Yaskawa INFORM job: A_ROOF_SIDE_0617_2_PAINT_20.JBI

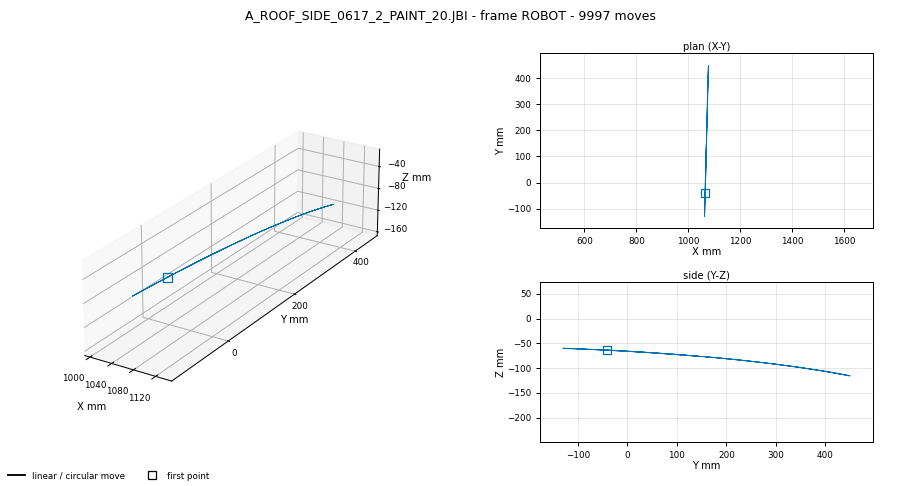
[picture p0: tool path of A_ROOF_SIDE_0617_2_PAINT_20.JBI in frame ROBOT, 9997 of 9997 moves have a stored position in this frame; points joined in program order, loops and branches not executed]
/JOB
//NAME A_ROOF_SIDE_0617_2_PAINT20
//POS
///NPOS 9997,0,0,0,0,0
///TOOL 1
///USER 0
///POSTYPE ROBOT
///RECTAN
///RCONF 1,0,0,0,0,0,0,0,0,0,0,0,0,0,0,0,0,0,0,0,0,0,0,0
C00000=1065.238,-41.066,-63.306,172.043,25.309,154.670
C00001=1065.244,-40.817,-63.319,172.044,25.312,154.670
C00002=1065.251,-40.567,-63.331,172.046,25.313,154.670
C00003=1065.257,-40.317,-63.343,172.047,25.316,154.670
C00004=1065.263,-40.068,-63.356,172.049,25.318,154.670
C00005=1065.269,-39.818,-63.369,172.050,25.320,154.671
C00006=1065.275,-39.568,-63.382,172.052,25.322,154.671
C00007=1065.281,-39.319,-63.394,172.053,25.324,154.671
C00008=1065.288,-39.070,-63.407,172.055,25.327,154.671
C00009=1065.294,-38.820,-63.420,172.056,25.328,154.671
C00010=1065.299,-38.570,-63.432,172.058,25.331,154.672
C00011=1065.305,-38.321,-63.445,172.059,25.332,154.672
C00012=1065.311,-38.071,-63.458,172.061,25.335,154.672
C00013=1065.317,-37.822,-63.471,172.063,25.337,154.672
C00014=1065.323,-37.572,-63.483,172.065,25.339,154.673
C00015=1065.329,-37.322,-63.496,172.066,25.342,154.673
C00016=1065.335,-37.073,-63.509,172.068,25.344,154.673
C00017=1065.341,-36.823,-63.522,172.069,25.346,154.673
C00018=1065.347,-36.573,-63.534,172.071,25.348,154.673
C00019=1065.353,-36.324,-63.548,172.072,25.350,154.674
C00020=1065.359,-36.074,-63.560,172.074,25.352,154.674
C00021=1065.365,-35.825,-63.573,172.075,25.355,154.674
C00022=1065.371,-35.575,-63.586,172.077,25.357,154.674
C00023=1065.378,-35.326,-63.599,172.078,25.359,154.675
C00024=1065.383,-35.076,-63.612,172.080,25.361,154.675
C00025=1065.390,-34.827,-63.625,172.081,25.363,154.675
C00026=1065.396,-34.577,-63.638,172.083,25.366,154.675
C00027=1065.402,-34.299,-63.652,172.084,25.368,154.676
C00028=1065.409,-34.021,-63.666,172.085,25.371,154.676
C00029=1065.416,-33.744,-63.680,172.088,25.373,154.676
C00030=1065.423,-33.466,-63.696,172.089,25.376,154.676
C00031=1065.429,-33.216,-63.708,172.091,25.377,154.677
C00032=1065.435,-32.967,-63.721,172.092,25.380,154.677
C00033=1065.441,-32.717,-63.734,172.094,25.382,154.677
C00034=1065.447,-32.468,-63.747,172.095,25.384,154.677
C00035=1065.453,-32.218,-63.760,172.097,25.386,154.677
C00036=1065.459,-31.969,-63.773,172.098,25.389,154.678
C00037=1065.465,-31.719,-63.786,172.100,25.391,154.678
C00038=1065.471,-31.470,-63.799,172.101,25.393,154.678
C00039=1065.477,-31.220,-63.811,172.103,25.395,154.678
C00040=1065.483,-30.970,-63.825,172.104,25.397,154.679
C00041=1065.490,-30.721,-63.838,172.106,25.400,154.679
C00042=1065.496,-30.471,-63.851,172.107,25.402,154.679
C00043=1065.502,-30.222,-63.864,172.109,25.404,154.679
C00044=1065.508,-29.971,-63.877,172.110,25.406,154.680
C00045=1065.514,-29.722,-63.890,172.112,25.409,154.680
C00046=1065.521,-29.473,-63.903,172.113,25.410,154.680
C00047=1065.526,-29.223,-63.916,172.115,25.413,154.680
C00048=1065.532,-28.973,-63.930,172.116,25.415,154.681
C00049=1065.538,-28.724,-63.943,172.117,25.417,154.681
C00050=1065.544,-28.474,-63.956,172.119,25.419,154.681
C00051=1065.550,-28.225,-63.969,172.121,25.422,154.681
C00052=1065.557,-27.976,-63.982,172.122,25.424,154.682
C00053=1065.563,-27.725,-63.995,172.123,25.426,154.682
C00054=1065.569,-27.476,-64.008,172.125,25.428,154.682
C00055=1065.576,-27.227,-64.022,172.126,25.430,154.682
C00056=1065.581,-26.977,-64.034,172.129,25.433,154.682
C00057=1065.588,-26.727,-64.047,172.130,25.435,154.683
C00058=1065.593,-26.478,-64.061,172.132,25.438,154.683
C00059=1065.599,-26.229,-64.074,172.133,25.440,154.683
C00060=1065.605,-25.979,-64.087,172.135,25.442,154.684
C00061=1065.611,-25.729,-64.101,172.136,25.444,154.684
C00062=1065.618,-25.479,-64.115,172.138,25.447,154.684
C00063=1065.624,-25.230,-64.128,172.139,25.449,154.684
C00064=1065.630,-24.980,-64.140,172.141,25.451,154.684
C00065=1065.635,-24.731,-64.154,172.142,25.454,154.685
C00066=1065.641,-24.481,-64.167,172.143,25.456,154.685
C00067=1065.648,-24.232,-64.181,172.145,25.458,154.685
C00068=1065.653,-23.982,-64.194,172.146,25.461,154.686
C00069=1065.659,-23.733,-64.207,172.148,25.463,154.686
C00070=1065.666,-23.483,-64.221,172.149,25.465,154.686
C00071=1065.671,-23.233,-64.235,172.151,25.468,154.686
C00072=1065.677,-22.984,-64.248,172.152,25.470,154.687
C00073=1065.684,-22.734,-64.261,172.154,25.472,154.687
C00074=1065.689,-22.484,-64.274,172.155,25.474,154.687
C00075=1065.695,-22.235,-64.288,172.157,25.477,154.687
C00076=1065.702,-21.985,-64.301,172.158,25.479,154.688
C00077=1065.707,-21.735,-64.315,172.160,25.481,154.688
C00078=1065.714,-21.486,-64.328,172.161,25.484,154.688
C00079=1065.720,-21.237,-64.342,172.163,25.486,154.688
C00080=1065.725,-20.987,-64.356,172.164,25.488,154.689
C00081=1065.731,-20.738,-64.369,172.165,25.491,154.689
C00082=1065.738,-20.488,-64.382,172.167,25.493,154.689
C00083=1065.743,-20.238,-64.396,172.168,25.495,154.689
C00084=1065.750,-19.989,-64.409,172.170,25.498,154.690
C00085=1065.756,-19.739,-64.422,172.171,25.500,154.690
C00086=1065.761,-19.490,-64.436,172.173,25.502,154.690
C00087=1065.768,-19.240,-64.450,172.174,25.505,154.691
C00088=1065.774,-18.991,-64.463,172.176,25.507,154.691
C00089=1065.780,-18.741,-64.477,172.177,25.509,154.691
C00090=1065.786,-18.492,-64.490,172.179,25.512,154.691
C00091=1065.793,-18.213,-64.505,172.180,25.514,154.692
C00092=1065.800,-17.934,-64.520,172.181,25.516,154.692
C00093=1065.807,-17.656,-64.536,172.184,25.520,154.692
C00094=1065.813,-17.377,-64.551,172.185,25.522,154.692
C00095=1065.820,-17.128,-64.565,172.187,25.524,154.693
C00096=1065.826,-16.879,-64.578,172.188,25.527,154.693
C00097=1065.832,-16.629,-64.592,172.190,25.529,154.693
C00098=1065.838,-16.379,-64.605,172.191,25.531,154.694
C00099=1065.844,-16.130,-64.619,172.192,25.534,154.694
C00100=1065.850,-15.881,-64.632,172.194,25.536,154.694
C00101=1065.857,-15.631,-64.646,172.195,25.538,154.694
C00102=1065.862,-15.381,-64.660,172.197,25.541,154.695
C00103=1065.868,-15.132,-64.673,172.198,25.543,154.695
C00104=1065.874,-14.881,-64.687,172.200,25.545,154.695
C00105=1065.881,-14.632,-64.701,172.201,25.548,154.695
C00106=1065.886,-14.383,-64.715,172.203,25.550,154.696
C00107=1065.893,-14.134,-64.729,172.204,25.552,154.696
C00108=1065.899,-13.884,-64.743,172.206,25.555,154.696
C00109=1065.904,-13.634,-64.757,172.207,25.557,154.697
C00110=1065.910,-13.385,-64.770,172.209,25.560,154.697
C00111=1065.916,-13.135,-64.784,172.210,25.562,154.697
C00112=1065.923,-12.885,-64.797,172.211,25.565,154.697
C00113=1065.928,-12.636,-64.811,172.213,25.567,154.698
C00114=1065.934,-12.387,-64.826,172.214,25.569,154.698
C00115=1065.940,-12.138,-64.839,172.216,25.572,154.698
C00116=1065.946,-11.887,-64.853,172.217,25.574,154.699
C00117=1065.953,-11.638,-64.867,172.219,25.576,154.699
C00118=1065.958,-11.388,-64.880,172.220,25.579,154.699
C00119=1065.964,-11.139,-64.895,172.221,25.582,154.699
C00120=1065.971,-10.889,-64.909,172.223,25.584,154.700
C00121=1065.976,-10.640,-64.923,172.224,25.586,154.700
C00122=1065.983,-10.390,-64.936,172.226,25.589,154.700
C00123=1065.988,-10.140,-64.950,172.227,25.591,154.701
C00124=1065.994,-9.891,-64.965,172.229,25.593,154.701
C00125=1066.001,-9.641,-64.978,172.230,25.596,154.701
C00126=1066.006,-9.392,-64.992,172.232,25.599,154.701
C00127=1066.012,-9.142,-65.006,172.233,25.601,154.702
C00128=1066.019,-8.893,-65.020,172.234,25.603,154.702
C00129=1066.025,-8.643,-65.034,172.236,25.606,154.702
C00130=1066.031,-8.394,-65.047,172.237,25.608,154.703
C00131=1066.037,-8.144,-65.062,172.239,25.610,154.703
C00132=1066.043,-7.895,-65.076,172.240,25.613,154.703
C00133=1066.049,-7.646,-65.090,172.242,25.616,154.703
C00134=1066.055,-7.396,-65.105,172.243,25.618,154.704
C00135=1066.061,-7.146,-65.118,172.245,25.620,154.704
C00136=1066.067,-6.896,-65.132,172.246,25.623,154.704
C00137=1066.073,-6.647,-65.147,172.247,25.625,154.705
C00138=1066.079,-6.398,-65.160,172.249,25.627,154.705
C00139=1066.086,-6.148,-65.174,172.250,25.630,154.705
C00140=1066.091,-5.899,-65.189,172.252,25.633,154.706
C00141=1066.097,-5.649,-65.203,172.253,25.635,154.706
C00142=1066.104,-5.399,-65.216,172.255,25.637,154.706
C00143=1066.110,-5.150,-65.231,172.256,25.640,154.706
C00144=1066.115,-4.900,-65.245,172.258,25.642,154.707
C00145=1066.122,-4.652,-65.259,172.259,25.644,154.707
C00146=1066.128,-4.401,-65.273,172.260,25.647,154.707
C00147=1066.134,-4.152,-65.287,172.262,25.649,154.708
C00148=1066.141,-3.902,-65.301,172.263,25.652,154.708
C00149=1066.146,-3.653,-65.315,172.265,25.654,154.708
C00150=1066.153,-3.403,-65.330,172.266,25.656,154.708
C00151=1066.158,-3.154,-65.344,172.268,25.659,154.709
C00152=1066.164,-2.905,-65.359,172.269,25.662,154.709
C00153=1066.171,-2.655,-65.372,172.271,25.664,154.709
C00154=1066.176,-2.405,-65.386,172.272,25.666,154.710
C00155=1066.182,-2.125,-65.403,172.273,25.669,154.710
C00156=1066.189,-1.844,-65.419,172.275,25.672,154.710
C00157=1066.196,-1.565,-65.435,172.277,25.675,154.711
C00158=1066.202,-1.285,-65.451,172.278,25.678,154.711
C00159=1066.208,-1.035,-65.465,172.280,25.681,154.711
C00160=1066.214,-0.786,-65.480,172.281,25.683,154.712
C00161=1066.220,-0.536,-65.494,172.283,25.685,154.712
C00162=1066.226,-0.286,-65.509,172.284,25.688,154.712
C00163=1066.232,-0.037,-65.523,172.286,25.691,154.713
C00164=1066.238,0.213,-65.538,172.287,25.693,154.713
C00165=1066.245,0.461,-65.552,172.288,25.696,154.713
C00166=1066.250,0.711,-65.566,172.290,25.698,154.713
C00167=1066.256,0.961,-65.581,172.291,25.700,154.714
C00168=1066.262,1.210,-65.595,172.293,25.703,154.714
C00169=1066.268,1.460,-65.610,172.294,25.706,154.714
C00170=1066.274,1.709,-65.624,172.296,25.708,154.715
C00171=1066.280,1.959,-65.638,172.297,25.711,154.715
C00172=1066.286,2.208,-65.653,172.298,25.713,154.715
C00173=1066.292,2.458,-65.667,172.300,25.716,154.716
C00174=1066.298,2.707,-65.682,172.301,25.719,154.716
C00175=1066.304,2.957,-65.697,172.303,25.721,154.716
C00176=1066.310,3.207,-65.711,172.304,25.723,154.717
C00177=1066.316,3.456,-65.725,172.305,25.726,154.717
C00178=1066.322,3.705,-65.740,172.307,25.728,154.717
C00179=1066.328,3.955,-65.754,172.308,25.731,154.717
C00180=1066.334,4.204,-65.769,172.310,25.734,154.718
C00181=1066.340,4.454,-65.784,172.311,25.736,154.718
C00182=1066.346,4.704,-65.798,172.313,25.738,154.718
C00183=1066.352,4.953,-65.813,172.314,25.741,154.719
C00184=1066.358,5.202,-65.827,172.316,25.744,154.719
C00185=1066.364,5.452,-65.842,172.317,25.746,154.719
C00186=1066.370,5.701,-65.856,172.318,25.749,154.720
C00187=1066.376,5.951,-65.871,172.320,25.751,154.720
C00188=1066.382,6.200,-65.886,172.320,25.754,154.720
C00189=1066.388,6.450,-65.900,172.322,25.756,154.721
C00190=1066.394,6.699,-65.914,172.323,25.758,154.721
C00191=1066.400,6.949,-65.929,172.325,25.761,154.721
C00192=1066.406,7.199,-65.944,172.326,25.764,154.722
C00193=1066.412,7.448,-65.959,172.328,25.766,154.722
C00194=1066.417,7.698,-65.974,172.329,25.769,154.722
C00195=1066.423,7.947,-65.988,172.330,25.771,154.723
C00196=1066.430,8.197,-66.003,172.332,25.773,154.723
C00197=1066.435,8.446,-66.018,172.333,25.776,154.723
C00198=1066.442,8.695,-66.033,172.335,25.779,154.724
C00199=1066.448,8.946,-66.047,172.336,25.781,154.724
C00200=1066.454,9.195,-66.062,172.337,25.784,154.724
C00201=1066.460,9.444,-66.076,172.339,25.786,154.725
C00202=1066.466,9.694,-66.091,172.340,25.789,154.725
C00203=1066.472,9.943,-66.106,172.342,25.791,154.725
C00204=1066.479,10.193,-66.121,172.343,25.794,154.725
C00205=1066.484,10.441,-66.136,172.345,25.797,154.726
C00206=1066.490,10.692,-66.150,172.346,25.799,154.726
C00207=1066.497,10.941,-66.165,172.348,25.801,154.726
C00208=1066.503,11.190,-66.179,172.349,25.804,154.727
C00209=1066.509,11.440,-66.194,172.350,25.807,154.727
C00210=1066.515,11.690,-66.209,172.352,25.809,154.727
C00211=1066.520,11.939,-66.224,172.353,25.812,154.728
C00212=1066.527,12.189,-66.239,172.355,25.814,154.728
C00213=1066.533,12.438,-66.254,172.356,25.816,154.728
C00214=1066.539,12.687,-66.269,172.358,25.819,154.729
C00215=1066.545,12.937,-66.284,172.359,25.822,154.729
C00216=1066.552,13.187,-66.299,172.360,25.824,154.729
C00217=1066.558,13.435,-66.313,172.362,25.827,154.730
C00218=1066.564,13.685,-66.328,172.363,25.829,154.730
C00219=1066.571,13.967,-66.345,172.365,25.832,154.730
C00220=1066.577,14.249,-66.362,172.366,25.835,154.731
C00221=1066.584,14.532,-66.378,172.368,25.838,154.731
C00222=1066.591,14.813,-66.396,172.370,25.841,154.731
C00223=1066.597,15.063,-66.411,172.371,25.843,154.732
C00224=1066.603,15.312,-66.426,172.373,25.846,154.732
C00225=1066.609,15.562,-66.441,172.374,25.849,154.732
C00226=1066.615,15.812,-66.456,172.375,25.851,154.733
C00227=1066.621,16.061,-66.471,172.377,25.854,154.733
C00228=1066.627,16.310,-66.486,172.378,25.856,154.733
C00229=1066.633,16.560,-66.501,172.380,25.859,154.734
C00230=1066.638,16.809,-66.516,172.381,25.861,154.734
C00231=1066.645,17.059,-66.531,172.382,25.864,154.734
C00232=1066.651,17.308,-66.546,172.384,25.867,154.735
C00233=1066.656,17.558,-66.561,172.385,25.869,154.735
C00234=1066.663,17.807,-66.576,172.387,25.872,154.735
C00235=1066.669,18.057,-66.591,172.388,25.875,154.736
C00236=1066.674,18.306,-66.607,172.390,25.877,154.736
C00237=1066.681,18.555,-66.622,172.391,25.880,154.736
C00238=1066.687,18.805,-66.637,172.392,25.882,154.737
C00239=1066.693,19.055,-66.652,172.393,25.885,154.737
C00240=1066.699,19.304,-66.667,172.394,25.887,154.737
C00241=1066.705,19.554,-66.682,172.396,25.890,154.738
C00242=1066.711,19.803,-66.698,172.397,25.892,154.738
C00243=1066.717,20.053,-66.713,172.399,25.895,154.738
C00244=1066.723,20.302,-66.728,172.400,25.897,154.739
C00245=1066.729,20.552,-66.743,172.401,25.900,154.739
C00246=1066.735,20.801,-66.758,172.403,25.903,154.739
C00247=1066.740,21.050,-66.774,172.404,25.906,154.740
C00248=1066.747,21.299,-66.789,172.406,25.908,154.740
C00249=1066.752,21.549,-66.804,172.407,25.911,154.740
C00250=1066.759,21.799,-66.819,172.409,25.913,154.741
C00251=1066.764,22.048,-66.835,172.410,25.916,154.741
C00252=1066.771,22.297,-66.850,172.411,25.918,154.741
C00253=1066.776,22.547,-66.866,172.413,25.921,154.742
C00254=1066.783,22.797,-66.881,172.414,25.923,154.742
C00255=1066.789,23.045,-66.896,172.416,25.926,154.742
C00256=1066.794,23.295,-66.912,172.417,25.929,154.743
C00257=1066.801,23.545,-66.927,172.419,25.932,154.743
C00258=1066.806,23.795,-66.942,172.420,25.934,154.743
C00259=1066.812,24.043,-66.957,172.421,25.937,154.744
C00260=1066.818,24.293,-66.973,172.423,25.940,154.744
C00261=1066.824,24.543,-66.988,172.424,25.942,154.744
C00262=1066.830,24.792,-67.004,172.426,25.945,154.745
C00263=1066.837,25.042,-67.019,172.427,25.947,154.745
C00264=1066.842,25.291,-67.034,172.428,25.950,154.745
C00265=1066.849,25.540,-67.050,172.430,25.952,154.746
C00266=1066.854,25.790,-67.065,172.431,25.955,154.746
C00267=1066.861,26.040,-67.080,172.433,25.958,154.746
C00268=1066.866,26.289,-67.097,172.434,25.960,154.747
C00269=1066.872,26.538,-67.111,172.436,25.963,154.747
C00270=1066.878,26.788,-67.127,172.437,25.966,154.747
C00271=1066.885,27.037,-67.142,172.438,25.968,154.748
C00272=1066.890,27.287,-67.158,172.440,25.971,154.748
C00273=1066.897,27.536,-67.174,172.441,25.974,154.749
C00274=1066.902,27.785,-67.189,172.443,25.976,154.749
C00275=1066.908,28.035,-67.205,172.444,25.979,154.749
C00276=1066.914,28.284,-67.220,172.446,25.981,154.749
C00277=1066.920,28.534,-67.236,172.446,25.984,154.750
C00278=1066.927,28.783,-67.251,172.447,25.986,154.750
C00279=1066.933,29.033,-67.267,172.449,25.989,154.751
C00280=1066.938,29.282,-67.283,172.450,25.992,154.751
C00281=1066.944,29.531,-67.298,172.452,25.994,154.751
C00282=1066.950,29.781,-67.314,172.453,25.997,154.752
C00283=1066.957,30.064,-67.331,172.455,26.000,154.752
C00284=1066.964,30.348,-67.350,172.457,26.003,154.752
C00285=1066.971,30.631,-67.367,172.458,26.006,154.753
C00286=1066.977,30.914,-67.385,172.459,26.009,154.753
C00287=1066.983,31.164,-67.400,172.461,26.012,154.754
C00288=1066.989,31.414,-67.417,172.462,26.014,154.754
C00289=1066.995,31.663,-67.433,172.464,26.017,154.754
C00290=1067.001,31.913,-67.448,172.465,26.020,154.755
C00291=1067.006,32.161,-67.464,172.467,26.022,154.755
C00292=1067.012,32.411,-67.479,172.468,26.025,154.755
C00293=1067.019,32.660,-67.495,172.469,26.028,154.756
C00294=1067.024,32.910,-67.510,172.471,26.030,154.756
C00295=1067.030,33.160,-67.527,172.472,26.033,154.756
C00296=1067.036,33.409,-67.543,172.474,26.035,154.757
C00297=1067.043,33.659,-67.558,172.475,26.038,154.757
C00298=1067.049,33.908,-67.574,172.476,26.041,154.757
C00299=1067.055,34.157,-67.590,172.478,26.043,154.758
C00300=1067.060,34.407,-67.606,172.479,26.046,154.758
C00301=1067.066,34.656,-67.621,172.481,26.049,154.758
C00302=1067.072,34.906,-67.637,172.482,26.052,154.759
C00303=1067.078,35.155,-67.653,172.484,26.054,154.759
C00304=1067.085,35.404,-67.669,172.485,26.057,154.759
C00305=1067.091,35.653,-67.685,172.486,26.060,154.760
C00306=1067.096,35.903,-67.701,172.488,26.062,154.760
C00307=1067.102,36.153,-67.717,172.489,26.065,154.761
C00308=1067.108,36.402,-67.733,172.491,26.068,154.761
C00309=1067.115,36.652,-67.748,172.492,26.070,154.761
C00310=1067.120,36.901,-67.764,172.494,26.073,154.762
C00311=1067.126,37.150,-67.780,172.495,26.075,154.762
C00312=1067.132,37.400,-67.796,172.496,26.078,154.762
C00313=1067.139,37.649,-67.812,172.498,26.081,154.763
C00314=1067.145,37.899,-67.828,172.499,26.083,154.763
C00315=1067.151,38.148,-67.844,172.501,26.086,154.763
C00316=1067.156,38.398,-67.860,172.502,26.089,154.764
C00317=1067.162,38.647,-67.876,172.503,26.091,154.764
C00318=1067.168,38.896,-67.892,172.504,26.094,154.764
C00319=1067.174,39.145,-67.908,172.505,26.097,154.765
C00320=1067.179,39.395,-67.924,172.507,26.099,154.765
C00321=1067.185,39.645,-67.940,172.508,26.102,154.766
C00322=1067.191,39.894,-67.956,172.510,26.105,154.766
C00323=1067.197,40.143,-67.972,172.511,26.107,154.766
C00324=1067.203,40.393,-67.989,172.512,26.110,154.767
C00325=1067.209,40.642,-68.005,172.514,26.113,154.767
C00326=1067.216,40.891,-68.021,172.515,26.115,154.767
C00327=1067.221,41.141,-68.036,172.517,26.118,154.768
C00328=1067.227,41.391,-68.052,172.518,26.121,154.768
C00329=1067.233,41.640,-68.069,172.520,26.123,154.768
C00330=1067.239,41.889,-68.085,172.521,26.126,154.769
C00331=1067.245,42.139,-68.101,172.522,26.129,154.769
C00332=1067.251,42.388,-68.117,172.524,26.131,154.769
C00333=1067.257,42.637,-68.134,172.525,26.134,154.770
C00334=1067.263,42.887,-68.150,172.527,26.137,154.770
C00335=1067.269,43.136,-68.166,172.528,26.139,154.771
C00336=1067.275,43.385,-68.182,172.530,26.142,154.771
C00337=1067.280,43.635,-68.198,172.531,26.145,154.771
C00338=1067.286,43.885,-68.214,172.532,26.148,154.772
C00339=1067.292,44.134,-68.231,172.534,26.150,154.772
C00340=1067.298,44.384,-68.247,172.535,26.153,154.772
C00341=1067.304,44.633,-68.264,172.537,26.156,154.773
C00342=1067.310,44.882,-68.280,172.538,26.159,154.773
C00343=1067.315,45.132,-68.296,172.539,26.161,154.773
C00344=1067.321,45.381,-68.312,172.541,26.164,154.774
C00345=1067.327,45.631,-68.329,172.542,26.167,154.774
C00346=1067.333,45.880,-68.346,172.544,26.170,154.775
C00347=1067.340,46.163,-68.364,172.545,26.173,154.775
C00348=1067.346,46.447,-68.383,172.546,26.175,154.775
C00349=1067.352,46.730,-68.402,172.548,26.179,154.776
C00350=1067.360,47.013,-68.420,172.550,26.182,154.776
C00351=1067.365,47.263,-68.437,172.551,26.185,154.777
C00352=1067.371,47.512,-68.453,172.553,26.187,154.777
C00353=1067.377,47.761,-68.470,172.554,26.190,154.777
C00354=1067.383,48.011,-68.486,172.556,26.193,154.778
C00355=1067.389,48.260,-68.502,172.557,26.196,154.778
C00356=1067.394,48.510,-68.519,172.559,26.198,154.778
C00357=1067.400,48.759,-68.535,172.560,26.201,154.779
C00358=1067.406,49.008,-68.551,172.561,26.204,154.779
C00359=1067.412,49.258,-68.568,172.563,26.207,154.780
C00360=1067.417,49.507,-68.585,172.563,26.209,154.780
C00361=1067.423,49.756,-68.602,172.565,26.211,154.780
C00362=1067.429,50.005,-68.618,172.566,26.214,154.781
C00363=1067.436,50.255,-68.634,172.567,26.217,154.781
C00364=1067.441,50.505,-68.651,172.569,26.220,154.781
C00365=1067.447,50.754,-68.668,172.570,26.222,154.782
C00366=1067.453,51.004,-68.684,172.572,26.225,154.782
C00367=1067.459,51.253,-68.701,172.573,26.228,154.783
C00368=1067.464,51.502,-68.718,172.575,26.230,154.783
C00369=1067.470,51.752,-68.734,172.576,26.233,154.783
C00370=1067.476,52.001,-68.750,172.577,26.236,154.784
C00371=1067.482,52.250,-68.766,172.579,26.239,154.784
C00372=1067.488,52.499,-68.784,172.580,26.241,154.784
C00373=1067.494,52.749,-68.801,172.582,26.244,154.785
C00374=1067.500,52.999,-68.817,172.583,26.247,154.785
C00375=1067.506,53.248,-68.833,172.584,26.250,154.786
C00376=1067.512,53.497,-68.851,172.586,26.252,154.786
C00377=1067.518,53.746,-68.867,172.587,26.255,154.786
C00378=1067.524,53.996,-68.883,172.589,26.258,154.787
C00379=1067.530,54.245,-68.899,172.590,26.260,154.787
C00380=1067.536,54.495,-68.917,172.592,26.263,154.787
C00381=1067.542,54.744,-68.934,172.593,26.266,154.788
C00382=1067.548,54.994,-68.950,172.594,26.269,154.788
C00383=1067.553,55.243,-68.967,172.596,26.271,154.788
C00384=1067.559,55.492,-68.984,172.597,26.274,154.789
C00385=1067.565,55.741,-69.000,172.599,26.277,154.789
C00386=1067.572,55.991,-69.017,172.600,26.279,154.789
C00387=1067.577,56.240,-69.034,172.602,26.282,154.790
C00388=1067.583,56.490,-69.050,172.603,26.285,154.790
C00389=1067.589,56.738,-69.067,172.604,26.288,154.791
C00390=1067.595,56.988,-69.084,172.606,26.290,154.791
C00391=1067.601,57.238,-69.101,172.607,26.293,154.791
C00392=1067.607,57.487,-69.118,172.609,26.296,154.792
C00393=1067.613,57.737,-69.135,172.610,26.298,154.792
C00394=1067.619,57.986,-69.151,172.612,26.301,154.792
C00395=1067.625,58.235,-69.168,172.613,26.304,154.793
C00396=1067.631,58.485,-69.185,172.615,26.306,154.793
C00397=1067.637,58.734,-69.202,172.616,26.309,154.793
C00398=1067.643,58.983,-69.218,172.617,26.312,154.794
C00399=1067.649,59.233,-69.236,172.619,26.314,154.794
C00400=1067.655,59.482,-69.253,172.620,26.317,154.795
C00401=1067.661,59.732,-69.269,172.622,26.320,154.795
C00402=1067.666,59.981,-69.286,172.623,26.322,154.795
C00403=1067.673,60.231,-69.303,172.625,26.325,154.796
C00404=1067.679,60.479,-69.320,172.626,26.328,154.796
C00405=1067.684,60.729,-69.337,172.627,26.330,154.796
C00406=1067.691,60.978,-69.354,172.629,26.333,154.797
C00407=1067.697,61.228,-69.370,172.630,26.336,154.797
C00408=1067.703,61.477,-69.388,172.632,26.338,154.797
C00409=1067.709,61.726,-69.404,172.633,26.341,154.798
C00410=1067.716,61.976,-69.422,172.635,26.344,154.798
C00411=1067.722,62.258,-69.441,172.636,26.347,154.799
C00412=1067.729,62.542,-69.460,172.637,26.349,154.799
C00413=1067.736,62.825,-69.480,172.640,26.353,154.799
C00414=1067.742,63.108,-69.499,172.641,26.355,154.800
C00415=1067.748,63.358,-69.516,172.643,26.358,154.800
C00416=1067.755,63.607,-69.533,172.644,26.361,154.801
C00417=1067.760,63.856,-69.550,172.645,26.363,154.801
C00418=1067.767,64.106,-69.567,172.647,26.366,154.801
C00419=1067.773,64.354,-69.584,172.648,26.369,154.802
C00420=1067.778,64.604,-69.601,172.650,26.371,154.802
C00421=1067.784,64.854,-69.618,172.651,26.374,154.802
C00422=1067.791,65.103,-69.635,172.653,26.377,154.803
C00423=1067.796,65.352,-69.652,172.654,26.380,154.803
C00424=1067.803,65.602,-69.670,172.655,26.382,154.803
C00425=1067.808,65.851,-69.687,172.657,26.385,154.804
C00426=1067.813,66.100,-69.704,172.658,26.388,154.804
C00427=1067.820,66.349,-69.721,172.660,26.391,154.805
C00428=1067.826,66.599,-69.739,172.661,26.393,154.805
C00429=1067.832,66.848,-69.755,172.663,26.396,154.805
C00430=1067.837,67.097,-69.773,172.664,26.399,154.806
C00431=1067.843,67.347,-69.791,172.665,26.402,154.806
C00432=1067.849,67.596,-69.807,172.667,26.404,154.806
C00433=1067.855,67.845,-69.825,172.668,26.407,154.807
C00434=1067.861,68.095,-69.842,172.670,26.410,154.807
C00435=1067.867,68.344,-69.859,172.671,26.412,154.808
C00436=1067.872,68.593,-69.876,172.673,26.415,154.808
C00437=1067.879,68.843,-69.894,172.674,26.418,154.808
C00438=1067.885,69.092,-69.911,172.675,26.420,154.809
C00439=1067.890,69.319,-69.927,172.677,26.423,154.809
C00440=1067.896,69.546,-69.943,172.677,26.425,154.809
C00441=1067.900,69.774,-69.959,172.679,26.428,154.810
C00442=1067.906,70.001,-69.974,172.680,26.430,154.810
C00443=1067.912,70.228,-69.990,172.682,26.433,154.810
C00444=1067.917,70.455,-70.006,172.683,26.435,154.811
C00445=1067.923,70.682,-70.022,172.685,26.438,154.811
C00446=1067.927,70.910,-70.038,172.685,26.440,154.811
C00447=1067.934,71.159,-70.055,172.687,26.443,154.812
C00448=1067.940,71.408,-70.073,172.688,26.445,154.812
C00449=1067.945,71.657,-70.090,172.690,26.448,154.813
C00450=1067.951,71.906,-70.108,172.691,26.451,154.813
C00451=1067.957,72.157,-70.125,172.693,26.453,154.813
C00452=1067.963,72.406,-70.142,172.694,26.456,154.814
C00453=1067.969,72.655,-70.160,172.695,26.459,154.814
C00454=1067.974,72.904,-70.178,172.697,26.462,154.814
C00455=1067.980,73.153,-70.195,172.698,26.464,154.815
C00456=1067.986,73.403,-70.213,172.700,26.467,154.815
C00457=1067.992,73.652,-70.230,172.702,26.470,154.815
C00458=1067.998,73.901,-70.248,172.704,26.473,154.816
C00459=1068.004,74.151,-70.266,172.705,26.476,154.816
C00460=1068.010,74.400,-70.283,172.706,26.478,154.817
C00461=1068.015,74.650,-70.300,172.708,26.481,154.817
C00462=1068.021,74.899,-70.318,172.709,26.484,154.817
C00463=1068.028,75.149,-70.335,172.711,26.487,154.818
C00464=1068.033,75.398,-70.353,172.712,26.489,154.818
C00465=1068.039,75.647,-70.370,172.714,26.492,154.818
C00466=1068.045,75.896,-70.388,172.715,26.495,154.819
C00467=1068.050,76.145,-70.406,172.716,26.498,154.819
C00468=1068.057,76.395,-70.424,172.718,26.500,154.819
C00469=1068.063,76.644,-70.441,172.719,26.503,154.820
C00470=1068.069,76.894,-70.459,172.721,26.505,154.820
C00471=1068.074,77.143,-70.476,172.722,26.508,154.821
C00472=1068.081,77.392,-70.494,172.724,26.511,154.821
C00473=1068.086,77.641,-70.512,172.725,26.513,154.821
C00474=1068.092,77.891,-70.531,172.727,26.516,154.822
C00475=1068.100,78.218,-70.553,172.728,26.520,154.822
C00476=1068.108,78.545,-70.577,172.730,26.523,154.823
C00477=1068.116,78.872,-70.600,172.732,26.527,154.823
C00478=1068.123,79.200,-70.623,172.734,26.530,154.824
C00479=1068.128,79.449,-70.641,172.735,26.533,154.824
C00480=1068.135,79.698,-70.659,172.737,26.536,154.825
C00481=1068.140,79.947,-70.677,172.738,26.538,154.825
C00482=1068.146,80.197,-70.695,172.739,26.541,154.825
C00483=1068.152,80.446,-70.712,172.741,26.544,154.826
C00484=1068.158,80.696,-70.730,172.742,26.547,154.826
C00485=1068.164,80.945,-70.748,172.744,26.550,154.826
C00486=1068.170,81.194,-70.766,172.746,26.553,154.827
C00487=1068.176,81.443,-70.784,172.748,26.555,154.827
C00488=1068.180,81.692,-70.802,172.749,26.558,154.827
C00489=1068.186,81.942,-70.820,172.750,26.561,154.828
C00490=1068.192,82.191,-70.838,172.752,26.564,154.828
C00491=1068.198,82.441,-70.856,172.753,26.567,154.829
C00492=1068.204,82.689,-70.874,172.755,26.569,154.829
C00493=1068.210,82.939,-70.892,172.756,26.572,154.829
C00494=1068.216,83.188,-70.909,172.758,26.574,154.830
C00495=1068.222,83.438,-70.927,172.759,26.577,154.830
C00496=1068.228,83.687,-70.946,172.761,26.580,154.831
C00497=1068.234,83.936,-70.964,172.762,26.582,154.831
C00498=1068.239,84.186,-70.982,172.763,26.585,154.831
C00499=1068.245,84.435,-71.000,172.765,26.588,154.832
C00500=1068.251,84.684,-71.018,172.766,26.591,154.832
C00501=1068.256,84.933,-71.036,172.768,26.594,154.832
C00502=1068.263,85.183,-71.054,172.769,26.596,154.833
C00503=1068.268,85.431,-71.072,172.771,26.599,154.833
C00504=1068.275,85.681,-71.090,172.772,26.602,154.834
C00505=1068.280,85.930,-71.108,172.774,26.605,154.834
C00506=1068.286,86.180,-71.126,172.775,26.607,154.834
C00507=1068.292,86.429,-71.145,172.776,26.610,154.835
C00508=1068.297,86.678,-71.162,172.778,26.612,154.835
C00509=1068.304,86.927,-71.181,172.779,26.615,154.835
C00510=1068.309,87.176,-71.199,172.781,26.618,154.836
C00511=1068.315,87.426,-71.217,172.782,26.620,154.836
C00512=1068.322,87.675,-71.235,172.784,26.623,154.837
C00513=1068.327,87.924,-71.253,172.785,26.626,154.837
C00514=1068.333,88.174,-71.271,172.787,26.628,154.837
C00515=1068.339,88.423,-71.290,172.788,26.631,154.838
C00516=1068.345,88.672,-71.307,172.790,26.634,154.838
C00517=1068.351,88.922,-71.326,172.792,26.637,154.838
C00518=1068.357,89.171,-71.344,172.793,26.639,154.839
C00519=1068.363,89.420,-71.362,172.795,26.642,154.839
C00520=1068.368,89.670,-71.381,172.796,26.645,154.839
C00521=1068.374,89.919,-71.398,172.798,26.648,154.840
C00522=1068.380,90.168,-71.417,172.799,26.650,154.840
C00523=1068.386,90.417,-71.435,172.801,26.653,154.841
C00524=1068.392,90.666,-71.453,172.802,26.656,154.841
C00525=1068.398,90.916,-71.471,172.804,26.658,154.841
C00526=1068.404,91.165,-71.490,172.805,26.661,154.842
C00527=1068.410,91.414,-71.508,172.807,26.664,154.842
C00528=1068.415,91.664,-71.527,172.808,26.667,154.842
C00529=1068.421,91.913,-71.545,172.809,26.669,154.843
C00530=1068.427,92.162,-71.564,172.811,26.672,154.843
C00531=1068.432,92.411,-71.582,172.812,26.674,154.844
C00532=1068.439,92.660,-71.600,172.814,26.677,154.844
C00533=1068.444,92.910,-71.620,172.815,26.680,154.844
C00534=1068.450,93.159,-71.637,172.817,26.683,154.845
C00535=1068.456,93.408,-71.656,172.818,26.686,154.845
C00536=1068.462,93.658,-71.674,172.819,26.689,154.846
C00537=1068.467,93.906,-71.693,172.822,26.691,154.846
C00538=1068.473,94.156,-71.712,172.823,26.694,154.846
C00539=1068.480,94.439,-71.732,172.825,26.697,154.847
C00540=1068.487,94.722,-71.753,172.826,26.700,154.847
C00541=1068.493,95.005,-71.774,172.829,26.703,154.847
C00542=1068.500,95.288,-71.795,172.830,26.706,154.848
C00543=1068.505,95.537,-71.814,172.831,26.709,154.848
C00544=1068.512,95.786,-71.832,172.833,26.712,154.849
C00545=1068.516,96.036,-71.851,172.834,26.715,154.849
C00546=1068.523,96.285,-71.869,172.836,26.717,154.849
C00547=1068.529,96.534,-71.888,172.837,26.720,154.850
C00548=1068.534,96.783,-71.906,172.839,26.723,154.850
C00549=1068.541,97.033,-71.925,172.840,26.725,154.851
C00550=1068.546,97.282,-71.944,172.842,26.728,154.851
C00551=1068.553,97.531,-71.963,172.844,26.731,154.851
C00552=1068.557,97.780,-71.981,172.845,26.734,154.852
C00553=1068.564,98.030,-71.999,172.847,26.736,154.852
C00554=1068.570,98.279,-72.019,172.848,26.739,154.852
C00555=1068.576,98.528,-72.037,172.850,26.742,154.853
C00556=1068.581,98.777,-72.055,172.851,26.744,154.853
C00557=1068.587,99.027,-72.074,172.853,26.747,154.854
C00558=1068.594,99.276,-72.093,172.854,26.750,154.854
C00559=1068.599,99.525,-72.112,172.856,26.752,154.854
C00560=1068.605,99.774,-72.130,172.857,26.755,154.855
C00561=1068.611,100.024,-72.149,172.859,26.758,154.855
C00562=1068.617,100.273,-72.167,172.860,26.761,154.855
C00563=1068.623,100.522,-72.187,172.862,26.763,154.856
C00564=1068.628,100.771,-72.205,172.863,26.766,154.856
C00565=1068.634,101.021,-72.224,172.865,26.769,154.856
C00566=1068.640,101.270,-72.242,172.867,26.772,154.857
C00567=1068.646,101.519,-72.261,172.868,26.775,154.857
C00568=1068.651,101.768,-72.280,172.870,26.777,154.858
C00569=1068.657,102.017,-72.299,172.871,26.780,154.858
C00570=1068.663,102.266,-72.318,172.873,26.782,154.858
C00571=1068.669,102.516,-72.337,172.874,26.785,154.859
C00572=1068.675,102.764,-72.356,172.876,26.788,154.859
C00573=1068.680,103.014,-72.375,172.877,26.791,154.860
C00574=1068.686,103.264,-72.393,172.879,26.793,154.860
C00575=1068.692,103.513,-72.412,172.880,26.796,154.860
C00576=1068.697,103.762,-72.431,172.881,26.799,154.861
C00577=1068.703,104.011,-72.450,172.884,26.802,154.861
C00578=1068.709,104.261,-72.469,172.885,26.805,154.861
C00579=1068.715,104.510,-72.488,172.887,26.807,154.862
C00580=1068.721,104.759,-72.507,172.888,26.810,154.862
C00581=1068.726,105.008,-72.526,172.890,26.813,154.863
C00582=1068.732,105.257,-72.545,172.891,26.815,154.863
C00583=1068.738,105.506,-72.564,172.893,26.818,154.863
C00584=1068.744,105.756,-72.583,172.894,26.820,154.864
C00585=1068.750,106.005,-72.602,172.896,26.823,154.864
C00586=1068.755,106.254,-72.621,172.897,26.826,154.864
C00587=1068.761,106.503,-72.640,172.898,26.829,154.865
C00588=1068.767,106.753,-72.659,172.901,26.832,154.865
C00589=1068.773,107.002,-72.678,172.902,26.834,154.865
C00590=1068.779,107.251,-72.697,172.904,26.837,154.866
C00591=1068.784,107.501,-72.717,172.905,26.840,154.866
C00592=1068.790,107.750,-72.736,172.907,26.843,154.867
C00593=1068.796,107.998,-72.755,172.908,26.845,154.867
C00594=1068.802,108.247,-72.774,172.910,26.848,154.867
C00595=1068.808,108.497,-72.793,172.911,26.851,154.868
C00596=1068.813,108.746,-72.813,172.913,26.853,154.868
C00597=1068.820,108.995,-72.831,172.914,26.856,154.868
C00598=1068.825,109.245,-72.850,172.917,26.859,154.869
C00599=1068.831,109.494,-72.870,172.918,26.862,154.869
C00600=1068.837,109.743,-72.889,172.919,26.864,154.870
C00601=1068.843,109.991,-72.908,172.921,26.867,154.870
C00602=1068.849,110.241,-72.927,172.922,26.869,154.870
C00603=1068.856,110.524,-72.949,172.924,26.872,154.871
C00604=1068.862,110.807,-72.971,172.926,26.876,154.871
C00605=1068.869,111.090,-72.993,172.928,26.879,154.872
C00606=1068.875,111.373,-73.015,172.930,26.882,154.872
C00607=1068.881,111.623,-73.034,172.931,26.885,154.872
C00608=1068.886,111.872,-73.053,172.933,26.887,154.873
C00609=1068.893,112.121,-73.072,172.934,26.890,154.873
C00610=1068.899,112.370,-73.092,172.936,26.893,154.874
C00611=1068.904,112.620,-73.111,172.937,26.895,154.874
C00612=1068.910,112.869,-73.130,172.939,26.898,154.874
C00613=1068.916,113.118,-73.149,172.940,26.901,154.875
C00614=1068.921,113.366,-73.169,172.943,26.903,154.875
C00615=1068.927,113.616,-73.188,172.944,26.906,154.875
C00616=1068.933,113.865,-73.207,172.946,26.909,154.876
C00617=1068.939,114.114,-73.227,172.947,26.912,154.876
C00618=1068.944,114.364,-73.247,172.949,26.914,154.876
C00619=1068.950,114.613,-73.266,172.950,26.917,154.877
C00620=1068.956,114.862,-73.286,172.952,26.920,154.877
C00621=1068.962,115.111,-73.305,172.953,26.923,154.878
C00622=1068.967,115.361,-73.324,172.955,26.926,154.878
C00623=1068.973,115.610,-73.344,172.957,26.928,154.878
C00624=1068.979,115.859,-73.364,172.958,26.931,154.879
C00625=1068.984,116.108,-73.382,172.960,26.934,154.879
C00626=1068.990,116.356,-73.402,172.961,26.936,154.880
C00627=1068.995,116.606,-73.422,172.963,26.939,154.880
C00628=1069.001,116.855,-73.442,172.964,26.942,154.880
C00629=1069.007,117.104,-73.461,172.966,26.945,154.881
C00630=1069.012,117.354,-73.481,172.968,26.948,154.881
C00631=1069.018,117.603,-73.501,172.970,26.951,154.882
C00632=1069.024,117.852,-73.520,172.971,26.953,154.882
C00633=1069.030,118.101,-73.540,172.973,26.956,154.882
C00634=1069.035,118.351,-73.560,172.974,26.959,154.883
C00635=1069.041,118.600,-73.580,172.976,26.961,154.883
C00636=1069.047,118.849,-73.599,172.977,26.964,154.883
C00637=1069.053,119.098,-73.619,172.979,26.967,154.884
C00638=1069.058,119.347,-73.638,172.981,26.969,154.884
C00639=1069.064,119.596,-73.658,172.982,26.972,154.885
C00640=1069.070,119.845,-73.677,172.984,26.975,154.885
C00641=1069.075,120.095,-73.698,172.985,26.978,154.885
C00642=1069.081,120.344,-73.717,172.987,26.981,154.886
C00643=1069.087,120.593,-73.737,172.988,26.984,154.886
C00644=1069.093,120.842,-73.756,172.991,26.986,154.886
C00645=1069.099,121.091,-73.776,172.992,26.989,154.887
C00646=1069.104,121.341,-73.795,172.994,26.992,154.887
C00647=1069.110,121.590,-73.816,172.995,26.994,154.888
C00648=1069.115,121.839,-73.835,172.997,26.997,154.888
C00649=1069.121,122.088,-73.855,172.998,26.999,154.888
C00650=1069.127,122.337,-73.875,173.001,27.003,154.889
C00651=1069.133,122.586,-73.894,173.002,27.005,154.889
C00652=1069.138,122.835,-73.915,173.003,27.008,154.889
C00653=1069.144,123.085,-73.934,173.005,27.010,154.890
C00654=1069.150,123.333,-73.954,173.006,27.013,154.890
C00655=1069.156,123.582,-73.974,173.008,27.016,154.891
C00656=1069.162,123.832,-73.993,173.010,27.019,154.891
C00657=1069.167,124.081,-74.014,173.012,27.022,154.891
C00658=1069.173,124.330,-74.034,173.013,27.024,154.892
C00659=1069.179,124.579,-74.053,173.015,27.027,154.892
C00660=1069.185,124.828,-74.073,173.016,27.030,154.892
C00661=1069.191,125.077,-74.093,173.018,27.033,154.893
C00662=1069.196,125.327,-74.113,173.020,27.035,154.893
C00663=1069.202,125.576,-74.133,173.022,27.038,154.894
C00664=1069.208,125.825,-74.153,173.023,27.041,154.894
C00665=1069.214,126.074,-74.173,173.025,27.043,154.894
C00666=1069.219,126.323,-74.193,173.026,27.046,154.895
C00667=1069.226,126.606,-74.216,173.029,27.049,154.895
C00668=1069.234,126.889,-74.238,173.030,27.052,154.895
C00669=1069.239,127.172,-74.260,173.032,27.055,154.896
C00670=1069.246,127.455,-74.283,173.034,27.058,154.896
C00671=1069.252,127.704,-74.304,173.035,27.061,154.897
C00672=1069.258,127.953,-74.324,173.038,27.064,154.897
C00673=1069.263,128.202,-74.343,173.039,27.066,154.897
C00674=1069.270,128.452,-74.364,173.041,27.069,154.898
C00675=1069.275,128.701,-74.384,173.042,27.072,154.898
C00676=1069.281,128.950,-74.404,173.044,27.074,154.898
C00677=1069.287,129.199,-74.424,173.046,27.077,154.899
C00678=1069.293,129.447,-74.444,173.048,27.080,154.899
C00679=1069.298,129.697,-74.464,173.049,27.083,154.900
C00680=1069.305,129.947,-74.484,173.051,27.085,154.900
C00681=1069.311,130.196,-74.504,173.052,27.088,154.900
C00682=1069.316,130.445,-74.525,173.055,27.091,154.901
C00683=1069.322,130.694,-74.545,173.056,27.093,154.901
C00684=1069.328,130.942,-74.565,173.058,27.096,154.901
C00685=1069.334,131.192,-74.585,173.059,27.099,154.902
C00686=1069.340,131.441,-74.605,173.061,27.101,154.902
C00687=1069.346,131.690,-74.625,173.063,27.104,154.902
C00688=1069.352,131.939,-74.645,173.065,27.107,154.903
C00689=1069.357,132.189,-74.666,173.066,27.109,154.903
C00690=1069.363,132.438,-74.685,173.068,27.112,154.904
C00691=1069.368,132.687,-74.706,173.069,27.114,154.904
C00692=1069.374,132.936,-74.726,173.071,27.118,154.904
C00693=1069.380,133.185,-74.747,173.073,27.120,154.905
C00694=1069.386,133.434,-74.767,173.074,27.123,154.905
C00695=1069.392,133.684,-74.787,173.076,27.125,154.905
C00696=1069.397,133.933,-74.808,173.077,27.128,154.906
C00697=1069.403,134.181,-74.828,173.080,27.131,154.906
C00698=1069.408,134.430,-74.849,173.081,27.134,154.907
C00699=1069.414,134.679,-74.869,173.083,27.136,154.907
C00700=1069.420,134.929,-74.890,173.084,27.139,154.907
C00701=1069.426,135.177,-74.910,173.087,27.142,154.908
C00702=1069.432,135.427,-74.931,173.088,27.145,154.908
C00703=1069.438,135.675,-74.951,173.090,27.148,154.908
C00704=1069.443,135.925,-74.971,173.091,27.150,154.909
C00705=1069.449,136.174,-74.991,173.093,27.153,154.909
C00706=1069.455,136.423,-75.012,173.095,27.156,154.910
C00707=1069.460,136.672,-75.033,173.097,27.159,154.910
C00708=1069.466,136.922,-75.053,173.098,27.161,154.910
C00709=1069.472,137.170,-75.074,173.100,27.164,154.911
C00710=1069.478,137.419,-75.094,173.102,27.167,154.911
C00711=1069.483,137.668,-75.115,173.104,27.169,154.911
C00712=1069.490,137.918,-75.135,173.105,27.172,154.912
C00713=1069.495,138.167,-75.156,173.107,27.174,154.912
C00714=1069.500,138.416,-75.176,173.109,27.178,154.913
C00715=1069.507,138.665,-75.197,173.111,27.180,154.913
C00716=1069.513,138.914,-75.218,173.112,27.183,154.913
C00717=1069.518,139.163,-75.238,173.114,27.185,154.914
C00718=1069.524,139.412,-75.258,173.116,27.188,154.914
C00719=1069.530,139.662,-75.279,173.117,27.191,154.914
C00720=1069.535,139.910,-75.300,173.119,27.194,154.915
C00721=1069.541,140.159,-75.320,173.121,27.196,154.915
C00722=1069.547,140.409,-75.341,173.123,27.199,154.915
C00723=1069.552,140.658,-75.362,173.124,27.202,154.916
C00724=1069.558,140.907,-75.383,173.126,27.205,154.916
C00725=1069.564,141.155,-75.403,173.127,27.207,154.917
C00726=1069.570,141.405,-75.424,173.130,27.210,154.917
C00727=1069.575,141.654,-75.445,173.131,27.213,154.917
C00728=1069.581,141.903,-75.466,173.133,27.216,154.918
C00729=1069.587,142.152,-75.486,173.134,27.218,154.918
C00730=1069.593,142.401,-75.507,173.137,27.222,154.919
C00731=1069.599,142.684,-75.531,173.138,27.224,154.919
C00732=1069.606,142.967,-75.554,173.141,27.227,154.919
C00733=1069.612,143.250,-75.578,173.142,27.230,154.920
C00734=1069.618,143.533,-75.602,173.144,27.234,154.920
C00735=1069.625,143.781,-75.623,173.146,27.237,154.921
C00736=1069.630,144.031,-75.643,173.148,27.239,154.921
C00737=1069.636,144.280,-75.664,173.150,27.242,154.921
C00738=1069.641,144.529,-75.685,173.151,27.245,154.922
C00739=1069.646,144.778,-75.706,173.153,27.247,154.922
C00740=1069.653,145.027,-75.727,173.155,27.250,154.922
C00741=1069.659,145.276,-75.748,173.157,27.253,154.923
C00742=1069.664,145.525,-75.769,173.158,27.255,154.923
C00743=1069.670,145.774,-75.790,173.160,27.258,154.924
C00744=1069.676,146.023,-75.811,173.162,27.261,154.924
C00745=1069.681,146.273,-75.832,173.164,27.264,154.924
C00746=1069.688,146.521,-75.853,173.165,27.266,154.925
C00747=1069.693,146.770,-75.873,173.168,27.269,154.925
C00748=1069.699,147.019,-75.895,173.169,27.272,154.925
C00749=1069.704,147.268,-75.915,173.171,27.274,154.926
C00750=1069.711,147.518,-75.937,173.172,27.277,154.926
C00751=1069.716,147.767,-75.958,173.175,27.280,154.927
C00752=1069.722,148.016,-75.979,173.176,27.283,154.927
C00753=1069.728,148.265,-75.999,173.178,27.285,154.927
C00754=1069.734,148.513,-76.020,173.180,27.288,154.928
C00755=1069.739,148.763,-76.041,173.182,27.291,154.928
C00756=1069.745,149.011,-76.063,173.183,27.294,154.928
C00757=1069.751,149.261,-76.084,173.186,27.297,154.929
C00758=1069.756,149.510,-76.105,173.187,27.299,154.929
C00759=1069.762,149.758,-76.126,173.189,27.302,154.929
C00760=1069.768,150.008,-76.147,173.190,27.305,154.930
C00761=1069.773,150.257,-76.168,173.193,27.308,154.930
C00762=1069.780,150.506,-76.190,173.194,27.310,154.931
C00763=1069.785,150.755,-76.210,173.196,27.313,154.931
C00764=1069.791,151.004,-76.232,173.198,27.316,154.931
C00765=1069.796,151.253,-76.254,173.200,27.319,154.932
C00766=1069.802,151.503,-76.275,173.201,27.321,154.932
C00767=1069.807,151.751,-76.296,173.204,27.324,154.933
C00768=1069.813,152.000,-76.317,173.205,27.327,154.933
C00769=1069.819,152.249,-76.339,173.207,27.329,154.933
C00770=1069.824,152.498,-76.360,173.209,27.332,154.934
C00771=1069.830,152.747,-76.381,173.211,27.335,154.934
C00772=1069.836,152.996,-76.403,173.212,27.338,154.934
C00773=1069.842,153.245,-76.424,173.215,27.341,154.935
C00774=1069.847,153.494,-76.445,173.216,27.343,154.935
C00775=1069.853,153.743,-76.466,173.218,27.346,154.935
C00776=1069.859,153.992,-76.488,173.220,27.349,154.936
C00777=1069.865,154.241,-76.509,173.222,27.352,154.936
C00778=1069.870,154.491,-76.530,173.223,27.354,154.937
C00779=1069.876,154.740,-76.552,173.226,27.357,154.937
C00780=1069.881,154.988,-76.573,173.227,27.360,154.937
C00781=1069.888,155.237,-76.595,173.229,27.363,154.938
C00782=1069.893,155.486,-76.616,173.231,27.366,154.938
C00783=1069.899,155.735,-76.638,173.233,27.368,154.938
C00784=1069.905,155.984,-76.658,173.234,27.371,154.939
C00785=1069.910,156.234,-76.681,173.237,27.374,154.939
C00786=1069.916,156.482,-76.702,173.238,27.376,154.940
C00787=1069.922,156.732,-76.724,173.239,27.379,154.940
C00788=1069.928,156.981,-76.745,173.242,27.382,154.940
C00789=1069.933,157.230,-76.767,173.244,27.384,154.941
C00790=1069.939,157.479,-76.789,173.245,27.387,154.941
C00791=1069.944,157.727,-76.810,173.247,27.390,154.941
C00792=1069.951,157.976,-76.832,173.249,27.393,154.942
C00793=1069.956,158.225,-76.853,173.250,27.396,154.942
C00794=1069.962,158.475,-76.875,173.253,27.399,154.943
C00795=1069.968,158.757,-76.899,173.255,27.402,154.943
C00796=1069.974,159.040,-76.924,173.257,27.405,154.943
C00797=1069.981,159.323,-76.948,173.259,27.408,154.944
C00798=1069.988,159.605,-76.973,173.262,27.411,154.944
C00799=1069.994,159.854,-76.995,173.263,27.414,154.945
C00800=1069.999,160.102,-77.016,173.265,27.416,154.945
C00801=1070.005,160.352,-77.038,173.267,27.419,154.945
C00802=1070.010,160.600,-77.060,173.269,27.422,154.946
C00803=1070.016,160.850,-77.081,173.270,27.425,154.946
C00804=1070.023,161.099,-77.103,173.273,27.428,154.947
C00805=1070.027,161.348,-77.125,173.274,27.430,154.947
C00806=1070.034,161.597,-77.146,173.277,27.433,154.947
C00807=1070.038,161.846,-77.168,173.278,27.436,154.948
C00808=1070.045,162.095,-77.190,173.280,27.439,154.948
C00809=1070.049,162.344,-77.212,173.282,27.442,154.948
C00810=1070.055,162.593,-77.234,173.284,27.444,154.949
C00811=1070.061,162.842,-77.256,173.286,27.448,154.949
C00812=1070.066,163.091,-77.278,173.288,27.450,154.950
C00813=1070.072,163.340,-77.300,173.289,27.453,154.950
C00814=1070.077,163.589,-77.322,173.291,27.456,154.950
C00815=1070.083,163.838,-77.343,173.293,27.459,154.951
C00816=1070.088,164.087,-77.365,173.294,27.462,154.951
C00817=1070.094,164.336,-77.388,173.297,27.465,154.952
C00818=1070.100,164.585,-77.410,173.298,27.467,154.952
C00819=1070.105,164.834,-77.432,173.301,27.470,154.952
C00820=1070.111,165.083,-77.453,173.302,27.473,154.953
C00821=1070.116,165.331,-77.476,173.304,27.476,154.953
C00822=1070.122,165.581,-77.498,173.306,27.479,154.954
C00823=1070.128,165.830,-77.520,173.308,27.482,154.954
C00824=1070.133,166.079,-77.542,173.310,27.485,154.954
C00825=1070.139,166.327,-77.564,173.312,27.488,154.955
C00826=1070.144,166.576,-77.586,173.313,27.490,154.955
C00827=1070.149,166.825,-77.608,173.316,27.493,154.956
C00828=1070.156,167.074,-77.630,173.317,27.496,154.956
C00829=1070.161,167.323,-77.652,173.320,27.499,154.956
C00830=1070.166,167.572,-77.674,173.321,27.501,154.957
C00831=1070.172,167.821,-77.697,173.324,27.504,154.957
C00832=1070.177,168.070,-77.719,173.325,27.507,154.958
C00833=1070.183,168.319,-77.741,173.327,27.510,154.958
C00834=1070.189,168.568,-77.763,173.329,27.513,154.958
C00835=1070.194,168.817,-77.785,173.331,27.516,154.959
C00836=1070.200,169.066,-77.808,173.333,27.519,154.959
C00837=1070.206,169.315,-77.830,173.335,27.521,154.960
C00838=1070.211,169.564,-77.852,173.337,27.524,154.960
C00839=1070.217,169.812,-77.874,173.339,27.527,154.960
C00840=1070.223,170.062,-77.896,173.340,27.530,154.961
C00841=1070.228,170.311,-77.919,173.343,27.533,154.961
C00842=1070.233,170.559,-77.941,173.344,27.535,154.961
C00843=1070.240,170.808,-77.963,173.347,27.538,154.962
C00844=1070.245,171.058,-77.986,173.348,27.541,154.962
C00845=1070.251,171.306,-78.009,173.351,27.544,154.963
C00846=1070.256,171.555,-78.030,173.352,27.547,154.963
C00847=1070.262,171.804,-78.053,173.355,27.550,154.963
C00848=1070.268,172.053,-78.075,173.356,27.553,154.964
C00849=1070.274,172.302,-78.097,173.359,27.556,154.964
C00850=1070.279,172.551,-78.119,173.360,27.558,154.965
C00851=1070.285,172.800,-78.142,173.362,27.561,154.965
C00852=1070.291,173.049,-78.164,173.364,27.564,154.965
C00853=1070.296,173.298,-78.187,173.366,27.566,154.966
C00854=1070.302,173.547,-78.209,173.368,27.569,154.966
C00855=1070.307,173.795,-78.231,173.370,27.572,154.966
C00856=1070.313,174.044,-78.254,173.372,27.575,154.967
C00857=1070.319,174.294,-78.276,173.374,27.578,154.967
C00858=1070.325,174.542,-78.299,173.376,27.581,154.968
C00859=1070.331,174.825,-78.324,173.378,27.584,154.968
C00860=1070.337,175.107,-78.350,173.380,27.587,154.969
C00861=1070.344,175.389,-78.375,173.382,27.590,154.969
C00862=1070.350,175.671,-78.400,173.385,27.593,154.969
C00863=1070.357,175.920,-78.423,173.387,27.596,154.970
C00864=1070.362,176.169,-78.446,173.389,27.599,154.970
C00865=1070.368,176.418,-78.468,173.390,27.602,154.970
C00866=1070.373,176.667,-78.491,173.393,27.605,154.971
C00867=1070.380,176.916,-78.513,173.394,27.608,154.971
C00868=1070.385,177.165,-78.536,173.397,27.611,154.972
C00869=1070.390,177.414,-78.558,173.398,27.613,154.972
C00870=1070.396,177.663,-78.581,173.401,27.616,154.972
C00871=1070.403,177.911,-78.603,173.403,27.619,154.973
C00872=1070.408,178.161,-78.626,173.405,27.622,154.973
C00873=1070.414,178.410,-78.649,173.407,27.625,154.974
C00874=1070.420,178.658,-78.672,173.409,27.627,154.974
C00875=1070.426,178.907,-78.694,173.411,27.630,154.974
C00876=1070.432,179.156,-78.717,173.413,27.633,154.975
C00877=1070.437,179.405,-78.739,173.415,27.636,154.975
C00878=1070.443,179.654,-78.762,173.417,27.638,154.975
C00879=1070.449,179.903,-78.785,173.419,27.641,154.976
C00880=1070.455,180.152,-78.807,173.421,27.644,154.976
C00881=1070.461,180.401,-78.830,173.423,27.647,154.977
C00882=1070.467,180.650,-78.853,173.425,27.650,154.977
C00883=1070.472,180.898,-78.876,173.427,27.652,154.977
C00884=1070.478,181.148,-78.898,173.429,27.655,154.978
C00885=1070.484,181.397,-78.921,173.431,27.658,154.978
C00886=1070.489,181.645,-78.943,173.433,27.661,154.978
C00887=1070.495,181.894,-78.966,173.435,27.664,154.979
C00888=1070.501,182.143,-78.989,173.437,27.667,154.979
C00889=1070.507,182.392,-79.013,173.439,27.669,154.980
C00890=1070.513,182.641,-79.035,173.442,27.672,154.980
C00891=1070.519,182.890,-79.058,173.443,27.675,154.980
C00892=1070.525,183.139,-79.081,173.446,27.678,154.981
C00893=1070.531,183.387,-79.104,173.447,27.681,154.981
C00894=1070.536,183.636,-79.127,173.450,27.684,154.981
C00895=1070.542,183.885,-79.150,173.451,27.686,154.982
C00896=1070.548,184.134,-79.173,173.454,27.689,154.982
C00897=1070.554,184.383,-79.195,173.455,27.691,154.983
C00898=1070.560,184.632,-79.218,173.458,27.695,154.983
C00899=1070.566,184.881,-79.241,173.460,27.698,154.983
C00900=1070.571,185.130,-79.264,173.462,27.700,154.984
C00901=1070.577,185.379,-79.287,173.464,27.703,154.984
C00902=1070.582,185.628,-79.310,173.466,27.706,154.985
C00903=1070.588,185.876,-79.333,173.468,27.709,154.985
C00904=1070.593,186.126,-79.357,173.470,27.712,154.985
C00905=1070.599,186.374,-79.380,173.472,27.715,154.986
C00906=1070.605,186.623,-79.403,173.474,27.718,154.986
C00907=1070.609,186.871,-79.426,173.476,27.721,154.987
C00908=1070.615,187.120,-79.449,173.479,27.724,154.987
C00909=1070.621,187.369,-79.472,173.480,27.727,154.987
C00910=1070.626,187.618,-79.495,173.483,27.730,154.988
C00911=1070.632,187.867,-79.520,173.484,27.733,154.988
C00912=1070.637,188.115,-79.543,173.487,27.736,154.989
C00913=1070.643,188.364,-79.565,173.489,27.739,154.989
C00914=1070.648,188.614,-79.589,173.491,27.741,154.989
C00915=1070.654,188.862,-79.612,173.493,27.745,154.990
C00916=1070.660,189.111,-79.636,173.495,27.748,154.990
C00917=1070.666,189.360,-79.659,173.497,27.751,154.991
C00918=1070.671,189.609,-79.682,173.499,27.753,154.991
C00919=1070.677,189.857,-79.706,173.501,27.756,154.992
C00920=1070.683,190.107,-79.729,173.504,27.759,154.992
C00921=1070.688,190.356,-79.753,173.505,27.762,154.992
C00922=1070.694,190.605,-79.776,173.508,27.765,154.993
C00923=1070.700,190.886,-79.803,173.510,27.769,154.993
C00924=1070.707,191.168,-79.829,173.512,27.772,154.994
C00925=1070.713,191.450,-79.855,173.515,27.775,154.994
C00926=1070.719,191.731,-79.882,173.517,27.779,154.995
C00927=1070.724,191.981,-79.905,173.519,27.781,154.995
C00928=1070.730,192.229,-79.929,173.521,27.784,154.995
C00929=1070.737,192.478,-79.952,173.524,27.787,154.996
C00930=1070.742,192.728,-79.976,173.525,27.790,154.996
C00931=1070.748,192.976,-79.999,173.528,27.793,154.997
C00932=1070.753,193.225,-80.022,173.529,27.796,154.997
C00933=1070.759,193.473,-80.047,173.532,27.799,154.997
C00934=1070.764,193.722,-80.070,173.534,27.802,154.998
C00935=1070.769,193.971,-80.093,173.536,27.805,154.998
C00936=1070.775,194.220,-80.117,173.538,27.808,154.999
C00937=1070.782,194.469,-80.140,173.541,27.811,154.999
C00938=1070.787,194.718,-80.164,173.542,27.814,154.999
C00939=1070.793,194.967,-80.187,173.545,27.817,155.000
C00940=1070.799,195.215,-80.211,173.547,27.820,155.000
C00941=1070.804,195.464,-80.235,173.549,27.823,155.001
C00942=1070.810,195.713,-80.258,173.551,27.826,155.001
C00943=1070.816,195.962,-80.283,173.553,27.828,155.001
C00944=1070.821,196.211,-80.306,173.555,27.831,155.002
C00945=1070.828,196.459,-80.329,173.558,27.834,155.002
C00946=1070.833,196.708,-80.353,173.559,27.837,155.003
C00947=1070.839,196.957,-80.377,173.562,27.840,155.003
C00948=1070.844,197.206,-80.401,173.564,27.844,155.004
C00949=1070.850,197.455,-80.424,173.566,27.846,155.004
C00950=1070.855,197.703,-80.448,173.568,27.849,155.004
C00951=1070.861,197.952,-80.471,173.571,27.852,155.005
C00952=1070.868,198.201,-80.495,173.572,27.855,155.005
C00953=1070.873,198.450,-80.520,173.575,27.858,155.006
C00954=1070.879,198.699,-80.543,173.577,27.861,155.006
C00955=1070.884,198.947,-80.567,173.580,27.864,155.006
C00956=1070.891,199.196,-80.591,173.581,27.867,155.007
C00957=1070.896,199.445,-80.614,173.584,27.870,155.007
C00958=1070.902,199.694,-80.638,173.586,27.873,155.007
C00959=1070.908,199.942,-80.662,173.588,27.875,155.008
C00960=1070.913,200.192,-80.686,173.590,27.878,155.008
C00961=1070.920,200.440,-80.709,173.592,27.882,155.009
C00962=1070.925,200.689,-80.734,173.594,27.885,155.009
C00963=1070.931,200.938,-80.758,173.597,27.888,155.010
C00964=1070.937,201.186,-80.782,173.599,27.891,155.010
C00965=1070.942,201.435,-80.805,173.601,27.893,155.010
C00966=1070.948,201.685,-80.829,173.603,27.896,155.011
C00967=1070.954,201.933,-80.853,173.606,27.899,155.011
C00968=1070.960,202.181,-80.877,173.608,27.902,155.012
C00969=1070.966,202.430,-80.901,173.610,27.905,155.012
C00970=1070.971,202.680,-80.925,173.612,27.908,155.012
C00971=1070.977,202.928,-80.949,173.614,27.912,155.013
C00972=1070.983,203.176,-80.973,173.616,27.914,155.013
C00973=1070.989,203.426,-80.998,173.618,27.917,155.014
C00974=1070.994,203.674,-81.022,173.621,27.920,155.014
C00975=1070.999,203.923,-81.046,173.623,27.924,155.015
C00976=1071.006,204.172,-81.070,173.625,27.927,155.015
C00977=1071.011,204.420,-81.094,173.627,27.930,155.015
C00978=1071.016,204.669,-81.119,173.630,27.933,155.016
C00979=1071.022,204.918,-81.143,173.632,27.936,155.016
C00980=1071.028,205.167,-81.167,173.634,27.939,155.017
C00981=1071.034,205.415,-81.191,173.636,27.942,155.017
C00982=1071.040,205.664,-81.216,173.639,27.945,155.017
C00983=1071.045,205.913,-81.240,173.640,27.948,155.018
C00984=1071.051,206.161,-81.264,173.643,27.951,155.018
C00985=1071.057,206.411,-81.288,173.645,27.954,155.019
C00986=1071.062,206.659,-81.313,173.648,27.957,155.019
C00987=1071.091,207.913,-81.436,173.784,28.030,155.022
C00988=1071.096,208.124,-81.456,173.785,28.033,155.023
C00989=1071.101,208.336,-81.478,173.787,28.037,155.023
C00990=1071.106,208.548,-81.499,173.789,28.040,155.024
C00991=1071.111,208.759,-81.521,173.791,28.043,155.024
C00992=1071.116,208.970,-81.541,173.792,28.047,155.025
C00993=1071.121,209.182,-81.563,173.795,28.050,155.025
C00994=1071.126,209.394,-81.584,173.796,28.054,155.026
C00995=1071.132,209.642,-81.609,173.798,28.058,155.026
C00996=1071.137,209.890,-81.634,173.800,28.061,155.027
C00997=1071.143,210.140,-81.659,173.802,28.065,155.028
C00998=1071.150,210.388,-81.684,173.804,28.069,155.028
C00999=1071.156,210.637,-81.710,173.806,28.073,155.029
C01000=1071.161,210.885,-81.735,173.808,28.077,155.030
C01001=1071.167,211.135,-81.760,173.810,28.081,155.030
C01002=1071.173,211.383,-81.785,173.812,28.085,155.031
C01003=1071.178,211.631,-81.810,173.814,28.089,155.032
C01004=1071.185,211.880,-81.836,173.817,28.093,155.032
C01005=1071.190,212.129,-81.860,173.819,28.097,155.033
C01006=1071.196,212.378,-81.886,173.820,28.101,155.033
C01007=1071.202,212.626,-81.911,173.823,28.105,155.034
C01008=1071.208,212.875,-81.936,173.825,28.109,155.035
C01009=1071.214,213.123,-81.962,173.826,28.113,155.035
C01010=1071.219,213.372,-81.988,173.829,28.117,155.036
C01011=1071.225,213.620,-82.013,173.831,28.121,155.037
C01012=1071.231,213.870,-82.037,173.833,28.125,155.037
C01013=1071.236,214.119,-82.063,173.835,28.129,155.038
C01014=1071.243,214.367,-82.089,173.837,28.133,155.039
C01015=1071.248,214.615,-82.114,173.839,28.137,155.039
C01016=1071.254,214.864,-82.139,173.841,28.141,155.040
C01017=1071.260,215.113,-82.165,173.843,28.145,155.041
C01018=1071.266,215.362,-82.190,173.846,28.149,155.041
C01019=1071.272,215.611,-82.216,173.848,28.153,155.042
C01020=1071.277,215.859,-82.241,173.849,28.157,155.042
C01021=1071.283,216.107,-82.266,173.852,28.161,155.043
C01022=1071.289,216.356,-82.292,173.854,28.165,155.044
C01023=1071.295,216.605,-82.318,173.856,28.169,155.044
C01024=1071.301,216.854,-82.343,173.858,28.173,155.045
C01025=1071.306,217.102,-82.369,173.860,28.177,155.046
C01026=1071.312,217.351,-82.394,173.862,28.181,155.046
C01027=1071.318,217.600,-82.420,173.865,28.185,155.047
C01028=1071.324,217.848,-82.445,173.866,28.188,155.047
C01029=1071.330,218.097,-82.471,173.869,28.192,155.048
C01030=1071.336,218.345,-82.497,173.871,28.196,155.049
C01031=1071.342,218.594,-82.523,173.873,28.200,155.049
C01032=1071.347,218.842,-82.548,173.875,28.204,155.050
C01033=1071.353,219.091,-82.573,173.877,28.208,155.051
C01034=1071.359,219.339,-82.599,173.879,28.212,155.051
C01035=1071.365,219.588,-82.625,173.882,28.216,155.052
C01036=1071.371,219.837,-82.650,173.883,28.220,155.053
C01037=1071.377,220.086,-82.677,173.886,28.224,155.053
C01038=1071.383,220.334,-82.702,173.888,28.228,155.054
C01039=1071.389,220.583,-82.728,173.890,28.231,155.054
C01040=1071.395,220.832,-82.753,173.892,28.235,155.055
C01041=1071.401,221.080,-82.779,173.894,28.239,155.056
C01042=1071.407,221.329,-82.805,173.896,28.243,155.056
C01043=1071.411,221.543,-82.827,173.898,28.247,155.057
C01044=1071.416,221.756,-82.849,173.900,28.250,155.057
C01045=1071.421,221.969,-82.872,173.902,28.253,155.058
C01046=1071.427,222.184,-82.894,173.903,28.257,155.058
C01047=1071.431,222.398,-82.916,173.906,28.261,155.059
C01048=1071.436,222.611,-82.938,173.907,28.264,155.060
C01049=1071.441,222.825,-82.960,173.910,28.267,155.060
C01050=1071.447,223.038,-82.983,173.911,28.271,155.061
C01051=1071.452,223.287,-83.009,173.914,28.275,155.061
C01052=1071.459,223.536,-83.035,173.916,28.279,155.062
C01053=1071.464,223.784,-83.061,173.917,28.282,155.063
C01054=1071.469,224.033,-83.087,173.920,28.286,155.063
C01055=1071.476,224.281,-83.113,173.922,28.290,155.064
C01056=1071.481,224.530,-83.139,173.924,28.294,155.065
C01057=1071.487,224.779,-83.165,173.927,28.298,155.065
C01058=1071.493,225.027,-83.191,173.928,28.302,155.066
C01059=1071.499,225.276,-83.217,173.931,28.306,155.066
C01060=1071.504,225.524,-83.243,173.933,28.310,155.067
C01061=1071.511,225.773,-83.269,173.935,28.314,155.068
C01062=1071.516,226.021,-83.295,173.938,28.318,155.068
C01063=1071.522,226.270,-83.321,173.939,28.322,155.069
C01064=1071.528,226.518,-83.348,173.942,28.326,155.070
C01065=1071.534,226.767,-83.373,173.944,28.330,155.070
C01066=1071.540,227.015,-83.400,173.946,28.334,155.071
C01067=1071.545,227.264,-83.426,173.949,28.338,155.072
C01068=1071.552,227.513,-83.452,173.950,28.341,155.072
C01069=1071.558,227.762,-83.478,173.952,28.345,155.073
C01070=1071.563,228.010,-83.505,173.955,28.349,155.073
C01071=1071.569,228.259,-83.531,173.957,28.353,155.074
C01072=1071.575,228.508,-83.557,173.960,28.357,155.075
C01073=1071.581,228.756,-83.583,173.961,28.361,155.075
C01074=1071.587,229.004,-83.610,173.963,28.365,155.076
C01075=1071.593,229.253,-83.635,173.966,28.368,155.076
C01076=1071.599,229.501,-83.662,173.968,28.372,155.077
C01077=1071.604,229.750,-83.688,173.971,28.376,155.078
C01078=1071.610,229.999,-83.715,173.973,28.380,155.078
C01079=1071.616,230.248,-83.742,173.974,28.384,155.079
C01080=1071.622,230.496,-83.768,173.977,28.388,155.080
C01081=1071.628,230.745,-83.794,173.979,28.392,155.080
C01082=1071.634,230.993,-83.820,173.982,28.396,155.081
C01083=1071.640,231.241,-83.847,173.984,28.400,155.082
C01084=1071.646,231.490,-83.874,173.986,28.404,155.082
C01085=1071.651,231.739,-83.900,173.988,28.407,155.083
C01086=1071.657,231.987,-83.926,173.990,28.411,155.083
C01087=1071.663,232.235,-83.953,173.993,28.415,155.084
C01088=1071.669,232.484,-83.979,173.995,28.419,155.085
C01089=1071.675,232.733,-84.006,173.997,28.423,155.085
C01090=1071.681,232.981,-84.033,174.000,28.427,155.086
C01091=1071.686,233.230,-84.059,174.002,28.431,155.087
C01092=1071.692,233.479,-84.086,174.004,28.435,155.087
C01093=1071.698,233.727,-84.112,174.006,28.439,155.088
C01094=1071.704,233.975,-84.139,174.008,28.443,155.089
C01095=1071.709,234.224,-84.166,174.011,28.447,155.089
C01096=1071.716,234.473,-84.193,174.013,28.451,155.090
C01097=1071.721,234.721,-84.219,174.016,28.455,155.090
C01098=1071.727,234.969,-84.246,174.018,28.459,155.091
C01099=1071.737,235.389,-84.291,174.021,28.465,155.092
C01100=1071.747,235.809,-84.336,174.025,28.472,155.093
C01101=1071.756,236.227,-84.381,174.029,28.479,155.094
C01102=1071.766,236.646,-84.426,174.033,28.485,155.095
C01103=1071.772,236.895,-84.453,174.035,28.489,155.096
C01104=1071.778,237.144,-84.480,174.038,28.493,155.097
C01105=1071.784,237.392,-84.507,174.040,28.497,155.097
C01106=1071.790,237.640,-84.533,174.042,28.501,155.098
C01107=1071.796,237.889,-84.560,174.044,28.504,155.098
C01108=1071.801,238.138,-84.588,174.046,28.508,155.099
C01109=1071.807,238.386,-84.614,174.049,28.512,155.100
C01110=1071.813,238.634,-84.642,174.051,28.516,155.100
C01111=1071.819,238.883,-84.668,174.054,28.520,155.101
C01112=1071.825,239.132,-84.695,174.056,28.524,155.102
C01113=1071.831,239.380,-84.722,174.058,28.528,155.102
C01114=1071.837,239.628,-84.749,174.061,28.532,155.103
C01115=1071.842,239.877,-84.776,174.063,28.536,155.103
C01116=1071.849,240.125,-84.804,174.065,28.540,155.104
C01117=1071.854,240.374,-84.830,174.067,28.544,155.105
C01118=1071.860,240.622,-84.857,174.070,28.548,155.105
C01119=1071.867,240.871,-84.884,174.072,28.552,155.106
C01120=1071.872,241.119,-84.912,174.074,28.556,155.107
C01121=1071.878,241.368,-84.939,174.077,28.559,155.107
C01122=1071.884,241.617,-84.966,174.079,28.563,155.108
C01123=1071.890,241.865,-84.992,174.082,28.567,155.108
C01124=1071.896,242.113,-85.020,174.084,28.571,155.109
C01125=1071.901,242.362,-85.047,174.086,28.575,155.110
C01126=1071.907,242.611,-85.074,174.089,28.579,155.110
C01127=1071.913,242.858,-85.101,174.091,28.583,155.111
C01128=1071.919,243.108,-85.129,174.093,28.587,155.112
C01129=1071.925,243.355,-85.156,174.095,28.590,155.112
C01130=1071.931,243.604,-85.183,174.098,28.594,155.113
C01131=1071.936,243.853,-85.210,174.100,28.598,155.113
C01132=1071.943,244.101,-85.238,174.102,28.602,155.114
C01133=1071.948,244.350,-85.265,174.105,28.606,155.115
C01134=1071.954,244.598,-85.293,174.107,28.610,155.115
C01135=1071.960,244.846,-85.319,174.110,28.614,155.116
C01136=1071.965,245.094,-85.347,174.112,28.618,155.117
C01137=1071.972,245.343,-85.374,174.114,28.622,155.117
C01138=1071.977,245.592,-85.402,174.117,28.626,155.118
C01139=1071.983,245.840,-85.429,174.119,28.630,155.119
C01140=1071.989,246.089,-85.457,174.122,28.634,155.119
C01141=1071.995,246.337,-85.484,174.124,28.638,155.120
C01142=1072.001,246.586,-85.512,174.127,28.642,155.120
C01143=1072.006,246.834,-85.539,174.129,28.646,155.121
C01144=1072.012,247.082,-85.567,174.130,28.649,155.122
C01145=1072.018,247.331,-85.595,174.133,28.653,155.122
C01146=1072.023,247.579,-85.622,174.135,28.657,155.123
C01147=1072.030,247.828,-85.650,174.138,28.661,155.124
C01148=1072.035,248.076,-85.678,174.140,28.665,155.124
C01149=1072.040,248.324,-85.705,174.143,28.669,155.125
C01150=1072.047,248.573,-85.733,174.145,28.673,155.126
C01151=1072.056,248.985,-85.779,174.149,28.680,155.127
C01152=1072.065,249.398,-85.825,174.153,28.686,155.128
C01153=1072.076,249.811,-85.871,174.157,28.693,155.129
C01154=1072.085,250.223,-85.917,174.161,28.700,155.130
C01155=1072.090,250.473,-85.945,174.164,28.704,155.131
C01156=1072.097,250.720,-85.972,174.166,28.708,155.131
C01157=1072.102,250.968,-86.000,174.168,28.712,155.132
C01158=1072.108,251.217,-86.028,174.171,28.716,155.133
C01159=1072.114,251.465,-86.056,174.173,28.720,155.133
C01160=1072.120,251.714,-86.084,174.176,28.724,155.134
C01161=1072.125,251.962,-86.111,174.178,28.728,155.134
C01162=1072.131,252.211,-86.140,174.181,28.731,155.135
C01163=1072.137,252.459,-86.167,174.183,28.735,155.136
C01164=1072.143,252.708,-86.195,174.185,28.739,155.136
C01165=1072.148,252.956,-86.223,174.188,28.743,155.137
C01166=1072.155,253.204,-86.251,174.190,28.747,155.138
C01167=1072.160,253.452,-86.279,174.193,28.751,155.138
C01168=1072.166,253.701,-86.307,174.195,28.755,155.139
C01169=1072.172,253.950,-86.336,174.198,28.759,155.139
C01170=1072.178,254.197,-86.363,174.200,28.763,155.140
C01171=1072.184,254.446,-86.391,174.202,28.767,155.141
C01172=1072.189,254.694,-86.419,174.205,28.771,155.141
C01173=1072.195,254.943,-86.448,174.207,28.775,155.142
C01174=1072.202,255.191,-86.475,174.210,28.779,155.143
C01175=1072.207,255.439,-86.503,174.212,28.782,155.143
C01176=1072.213,255.688,-86.532,174.215,28.786,155.144
C01177=1072.219,255.936,-86.560,174.217,28.790,155.145
C01178=1072.225,256.185,-86.587,174.220,28.794,155.145
C01179=1072.231,256.433,-86.615,174.222,28.798,155.146
C01180=1072.237,256.682,-86.644,174.224,28.802,155.146
C01181=1072.243,256.930,-86.672,174.227,28.806,155.147
C01182=1072.248,257.178,-86.701,174.229,28.810,155.148
C01183=1072.255,257.426,-86.728,174.232,28.814,155.148
C01184=1072.261,257.675,-86.757,174.234,28.817,155.149
C01185=1072.266,257.923,-86.785,174.237,28.821,155.150
C01186=1072.272,258.172,-86.813,174.239,28.825,155.150
C01187=1072.278,258.420,-86.841,174.242,28.829,155.151
C01188=1072.285,258.668,-86.869,174.244,28.833,155.152
C01189=1072.290,258.916,-86.898,174.246,28.837,155.152
C01190=1072.296,259.165,-86.926,174.249,28.841,155.153
C01191=1072.302,259.413,-86.954,174.252,28.845,155.153
C01192=1072.308,259.661,-86.983,174.255,28.849,155.154
C01193=1072.315,259.910,-87.011,174.257,28.853,155.155
C01194=1072.320,260.158,-87.039,174.260,28.857,155.155
C01195=1072.326,260.406,-87.067,174.262,28.860,155.156
C01196=1072.332,260.655,-87.096,174.265,28.864,155.157
C01197=1072.338,260.903,-87.124,174.267,28.868,155.157
C01198=1072.344,261.151,-87.152,174.270,28.872,155.158
C01199=1072.350,261.400,-87.181,174.272,28.876,155.158
C01200=1072.356,261.648,-87.209,174.274,28.880,155.159
C01201=1072.363,261.896,-87.238,174.277,28.884,155.160
C01202=1072.369,262.145,-87.266,174.279,28.888,155.160
C01203=1072.378,262.555,-87.313,174.283,28.894,155.161
C01204=1072.389,262.965,-87.360,174.289,28.900,155.162
C01205=1072.398,263.375,-87.408,174.293,28.907,155.163
C01206=1072.408,263.786,-87.454,174.297,28.913,155.164
C01207=1072.414,264.034,-87.483,174.299,28.917,155.165
C01208=1072.420,264.282,-87.512,174.302,28.921,155.166
C01209=1072.426,264.531,-87.541,174.304,28.925,155.166
C01210=1072.432,264.778,-87.569,174.307,28.929,155.167
C01211=1072.438,265.027,-87.598,174.309,28.933,155.168
C01212=1072.443,265.275,-87.627,174.311,28.937,155.168
C01213=1072.449,265.524,-87.656,174.314,28.941,155.169
C01214=1072.455,265.772,-87.685,174.316,28.945,155.170
C01215=1072.461,266.019,-87.713,174.320,28.949,155.170
C01216=1072.467,266.268,-87.742,174.322,28.953,155.171
C01217=1072.472,266.517,-87.771,174.325,28.957,155.171
C01218=1072.479,266.765,-87.800,174.327,28.961,155.172
C01219=1072.485,267.014,-87.829,174.330,28.965,155.173
C01220=1072.490,267.261,-87.857,174.332,28.969,155.173
C01221=1072.497,267.509,-87.887,174.335,28.973,155.174
C01222=1072.502,267.758,-87.916,174.337,28.976,155.175
C01223=1072.508,268.006,-87.944,174.339,28.980,155.175
C01224=1072.514,268.254,-87.974,174.343,28.985,155.176
C01225=1072.521,268.503,-88.003,174.345,28.989,155.177
C01226=1072.527,268.751,-88.032,174.348,28.992,155.177
C01227=1072.531,268.999,-88.060,174.350,28.996,155.178
C01228=1072.538,269.247,-88.089,174.353,29.000,155.179
C01229=1072.544,269.495,-88.118,174.355,29.004,155.179
C01230=1072.549,269.744,-88.148,174.358,29.008,155.180
C01231=1072.556,269.992,-88.177,174.360,29.012,155.181
C01232=1072.562,270.240,-88.206,174.364,29.016,155.181
C01233=1072.567,270.488,-88.236,174.366,29.020,155.182
C01234=1072.573,270.737,-88.264,174.368,29.024,155.182
C01235=1072.579,270.985,-88.293,174.371,29.028,155.183
C01236=1072.584,271.233,-88.322,174.373,29.032,155.184
C01237=1072.591,271.481,-88.351,174.376,29.036,155.184
C01238=1072.597,271.729,-88.380,174.378,29.040,155.185
C01239=1072.602,271.978,-88.410,174.382,29.044,155.186
C01240=1072.609,272.226,-88.439,174.384,29.048,155.186
C01241=1072.614,272.474,-88.469,174.387,29.052,155.187
C01242=1072.621,272.723,-88.498,174.389,29.056,155.188
C01243=1072.627,272.971,-88.527,174.392,29.060,155.188
C01244=1072.632,273.219,-88.556,174.394,29.064,155.189
C01245=1072.639,273.467,-88.585,174.398,29.068,155.190
C01246=1072.644,273.716,-88.615,174.400,29.072,155.190
C01247=1072.651,273.963,-88.645,174.403,29.076,155.191
C01248=1072.656,274.212,-88.674,174.405,29.080,155.192
C01249=1072.662,274.460,-88.703,174.407,29.084,155.192
C01250=1072.668,274.708,-88.733,174.410,29.088,155.193
C01251=1072.674,274.956,-88.762,174.413,29.092,155.194
C01252=1072.680,275.205,-88.792,174.416,29.096,155.194
C01253=1072.686,275.453,-88.821,174.418,29.100,155.195
C01254=1072.692,275.701,-88.851,174.421,29.104,155.196
C01255=1072.702,276.114,-88.899,174.425,29.111,155.197
C01256=1072.711,276.528,-88.949,174.430,29.117,155.198
C01257=1072.720,276.941,-88.998,174.434,29.124,155.199
C01258=1072.731,277.355,-89.048,174.438,29.130,155.200
C01259=1072.737,277.603,-89.077,174.442,29.135,155.201
C01260=1072.743,277.851,-89.108,174.444,29.139,155.201
C01261=1072.749,278.099,-89.137,174.447,29.143,155.202
C01262=1072.754,278.348,-89.166,174.449,29.147,155.203
C01263=1072.761,278.595,-89.196,174.452,29.151,155.203
C01264=1072.766,278.843,-89.226,174.455,29.155,155.204
C01265=1072.772,279.092,-89.255,174.457,29.159,155.205
C01266=1072.778,279.339,-89.285,174.460,29.163,155.205
C01267=1072.784,279.588,-89.315,174.462,29.167,155.206
C01268=1072.790,279.836,-89.345,174.465,29.171,155.207
C01269=1072.796,280.084,-89.374,174.468,29.175,155.207
C01270=1072.802,280.332,-89.405,174.471,29.179,155.208
C01271=1072.808,280.581,-89.435,174.473,29.183,155.209
C01272=1072.814,280.828,-89.464,174.476,29.187,155.209
C01273=1072.820,281.077,-89.494,174.479,29.191,155.210
C01274=1072.826,281.325,-89.524,174.482,29.195,155.211
C01275=1072.831,281.573,-89.554,174.484,29.200,155.211
C01276=1072.837,281.821,-89.584,174.487,29.203,155.212
C01277=1072.843,282.069,-89.614,174.489,29.207,155.213
C01278=1072.849,282.317,-89.644,174.493,29.211,155.213
C01279=1072.855,282.565,-89.673,174.495,29.216,155.214
C01280=1072.861,282.814,-89.704,174.498,29.220,155.215
C01281=1072.867,283.062,-89.734,174.500,29.224,155.215
C01282=1072.872,283.310,-89.764,174.503,29.228,155.216
C01283=1072.878,283.558,-89.794,174.506,29.232,155.217
C01284=1072.884,283.806,-89.825,174.508,29.236,155.217
C01285=1072.890,284.054,-89.854,174.511,29.240,155.218
C01286=1072.896,284.302,-89.884,174.514,29.244,155.219
C01287=1072.903,284.550,-89.915,174.517,29.248,155.219
C01288=1072.908,284.798,-89.945,174.519,29.253,155.220
C01289=1072.914,285.046,-89.975,174.522,29.257,155.221
C01290=1072.920,285.294,-90.005,174.525,29.261,155.221
C01291=1072.926,285.542,-90.036,174.528,29.265,155.222
C01292=1072.932,285.791,-90.066,174.530,29.268,155.223
C01293=1072.938,286.038,-90.097,174.533,29.273,155.223
C01294=1072.943,286.287,-90.126,174.536,29.277,155.224
C01295=1072.949,286.535,-90.157,174.539,29.281,155.225
C01296=1072.956,286.783,-90.187,174.541,29.285,155.225
C01297=1072.962,287.031,-90.217,174.545,29.289,155.226
C01298=1072.968,287.278,-90.247,174.547,29.293,155.227
C01299=1072.974,287.526,-90.278,174.550,29.297,155.227
C01300=1072.980,287.775,-90.309,174.552,29.301,155.228
C01301=1072.986,288.023,-90.339,174.556,29.305,155.229
C01302=1072.992,288.270,-90.369,174.558,29.310,155.230
C01303=1072.998,288.520,-90.399,174.560,29.314,155.230
C01304=1073.004,288.767,-90.430,174.564,29.318,155.231
C01305=1073.010,289.015,-90.460,174.566,29.322,155.231
C01306=1073.015,289.263,-90.490,174.569,29.326,155.232
C01307=1073.021,289.475,-90.517,174.571,29.329,155.233
C01308=1073.026,289.687,-90.543,174.574,29.333,155.233
C01309=1073.030,289.898,-90.569,174.577,29.337,155.234
C01310=1073.036,290.110,-90.596,174.578,29.340,155.235
C01311=1073.041,290.322,-90.621,174.581,29.344,155.235
C01312=1073.046,290.535,-90.647,174.583,29.347,155.236
C01313=1073.051,290.746,-90.674,174.586,29.350,155.236
C01314=1073.056,290.957,-90.699,174.588,29.354,155.237
C01315=1073.062,291.206,-90.731,174.591,29.358,155.238
C01316=1073.068,291.454,-90.761,174.593,29.362,155.238
C01317=1073.074,291.701,-90.792,174.597,29.367,155.239
C01318=1073.080,291.950,-90.823,174.599,29.371,155.240
C01319=1073.086,292.197,-90.853,174.602,29.375,155.240
C01320=1073.091,292.446,-90.884,174.605,29.379,155.241
C01321=1073.098,292.694,-90.915,174.608,29.383,155.242
C01322=1073.104,292.941,-90.946,174.610,29.387,155.243
C01323=1073.110,293.189,-90.976,174.614,29.392,155.243
C01324=1073.116,293.438,-91.007,174.616,29.395,155.244
C01325=1073.121,293.686,-91.038,174.619,29.400,155.245
C01326=1073.128,293.934,-91.069,174.622,29.404,155.245
C01327=1073.134,294.182,-91.100,174.625,29.408,155.246
C01328=1073.139,294.429,-91.130,174.627,29.412,155.247
C01329=1073.145,294.678,-91.162,174.631,29.416,155.247
C01330=1073.151,294.925,-91.192,174.633,29.421,155.248
C01331=1073.158,295.174,-91.223,174.636,29.425,155.249
C01332=1073.164,295.421,-91.254,174.639,29.429,155.250
C01333=1073.169,295.670,-91.285,174.642,29.433,155.250
C01334=1073.176,295.917,-91.316,174.645,29.437,155.251
C01335=1073.181,296.165,-91.347,174.647,29.442,155.252
C01336=1073.187,296.413,-91.379,174.650,29.446,155.252
C01337=1073.193,296.661,-91.409,174.653,29.450,155.253
C01338=1073.200,296.910,-91.440,174.656,29.454,155.254
C01339=1073.205,297.157,-91.472,174.658,29.459,155.254
C01340=1073.211,297.406,-91.502,174.662,29.463,155.255
C01341=1073.217,297.653,-91.534,174.664,29.467,155.256
C01342=1073.224,297.901,-91.565,174.667,29.471,155.257
C01343=1073.229,298.149,-91.596,174.670,29.476,155.257
C01344=1073.235,298.396,-91.627,174.673,29.480,155.258
C01345=1073.240,298.645,-91.659,174.676,29.484,155.259
C01346=1073.246,298.893,-91.690,174.679,29.488,155.260
C01347=1073.253,299.141,-91.722,174.681,29.493,155.260
C01348=1073.258,299.389,-91.753,174.685,29.497,155.261
C01349=1073.264,299.637,-91.784,174.687,29.501,155.262
C01350=1073.270,299.884,-91.816,174.690,29.506,155.262
C01351=1073.275,300.133,-91.847,174.693,29.510,155.263
C01352=1073.282,300.380,-91.878,174.696,29.514,155.264
C01353=1073.287,300.628,-91.910,174.699,29.519,155.265
C01354=1073.293,300.876,-91.942,174.702,29.523,155.265
C01355=1073.299,301.124,-91.973,174.704,29.527,155.266
C01356=1073.305,301.372,-92.004,174.708,29.532,155.267
C01357=1073.311,301.620,-92.036,174.710,29.536,155.268
C01358=1073.317,301.867,-92.067,174.714,29.540,155.268
C01359=1073.323,302.116,-92.099,174.716,29.545,155.269
C01360=1073.328,302.364,-92.130,174.720,29.549,155.270
C01361=1073.335,302.612,-92.162,174.722,29.553,155.271
C01362=1073.340,302.859,-92.193,174.724,29.557,155.271
C01363=1073.346,303.079,-92.222,174.727,29.561,155.272
C01364=1073.350,303.298,-92.249,174.730,29.565,155.272
C01365=1073.356,303.516,-92.278,174.732,29.569,155.273
C01366=1073.361,303.736,-92.306,174.736,29.573,155.274
C01367=1073.366,303.955,-92.334,174.738,29.576,155.274
C01368=1073.371,304.174,-92.362,174.741,29.580,155.275
C01369=1073.377,304.393,-92.390,174.743,29.584,155.276
C01370=1073.382,304.612,-92.417,174.746,29.588,155.276
C01371=1073.388,304.860,-92.449,174.748,29.592,155.277
C01372=1073.394,305.108,-92.481,174.752,29.597,155.278
C01373=1073.400,305.356,-92.513,174.754,29.601,155.279
C01374=1073.407,305.604,-92.544,174.757,29.605,155.279
C01375=1073.412,305.851,-92.576,174.760,29.609,155.280
C01376=1073.418,306.099,-92.608,174.763,29.614,155.281
C01377=1073.424,306.347,-92.640,174.766,29.618,155.282
C01378=1073.430,306.594,-92.672,174.769,29.623,155.282
C01379=1073.436,306.843,-92.704,174.772,29.627,155.283
C01380=1073.442,307.091,-92.736,174.775,29.631,155.284
C01381=1073.448,307.338,-92.767,174.778,29.636,155.285
C01382=1073.454,307.586,-92.799,174.781,29.640,155.285
C01383=1073.461,307.834,-92.831,174.784,29.644,155.286
C01384=1073.467,308.082,-92.863,174.787,29.649,155.287
C01385=1073.472,308.330,-92.895,174.790,29.653,155.288
C01386=1073.479,308.577,-92.927,174.793,29.658,155.288
C01387=1073.485,308.826,-92.959,174.796,29.662,155.289
C01388=1073.491,309.073,-92.991,174.799,29.666,155.290
C01389=1073.496,309.321,-93.023,174.802,29.671,155.291
C01390=1073.502,309.569,-93.055,174.805,29.675,155.291
C01391=1073.509,309.817,-93.086,174.808,29.679,155.292
C01392=1073.515,310.064,-93.119,174.811,29.683,155.293
C01393=1073.521,310.313,-93.151,174.814,29.688,155.294
C01394=1073.527,310.561,-93.183,174.817,29.692,155.294
C01395=1073.533,310.808,-93.216,174.820,29.696,155.295
C01396=1073.539,311.056,-93.248,174.823,29.701,155.296
C01397=1073.546,311.303,-93.280,174.826,29.705,155.297
C01398=1073.552,311.551,-93.312,174.829,29.710,155.297
C01399=1073.558,311.800,-93.344,174.832,29.714,155.298
C01400=1073.564,312.047,-93.377,174.835,29.718,155.299
C01401=1073.570,312.295,-93.409,174.838,29.723,155.300
C01402=1073.576,312.542,-93.441,174.841,29.727,155.300
C01403=1073.582,312.791,-93.473,174.844,29.732,155.301
C01404=1073.589,313.038,-93.505,174.847,29.736,155.302
C01405=1073.595,313.286,-93.537,174.850,29.741,155.303
C01406=1073.601,313.534,-93.570,174.853,29.745,155.303
C01407=1073.607,313.782,-93.602,174.856,29.749,155.304
C01408=1073.614,314.029,-93.635,174.860,29.754,155.305
C01409=1073.620,314.278,-93.667,174.862,29.758,155.306
C01410=1073.626,314.525,-93.699,174.866,29.763,155.306
C01411=1073.632,314.773,-93.732,174.868,29.767,155.307
C01412=1073.637,315.021,-93.765,174.872,29.772,155.308
C01413=1073.644,315.269,-93.798,174.874,29.776,155.309
C01414=1073.650,315.517,-93.830,174.878,29.781,155.310
C01415=1073.655,315.764,-93.862,174.880,29.785,155.310
C01416=1073.661,316.012,-93.895,174.884,29.790,155.311
C01417=1073.667,316.260,-93.928,174.886,29.794,155.312
C01418=1073.674,316.507,-93.961,174.890,29.799,155.313
C01419=1073.678,316.729,-93.990,174.892,29.803,155.314
C01420=1073.683,316.950,-94.019,174.895,29.807,155.314
C01421=1073.689,317.170,-94.048,174.897,29.812,155.315
C01422=1073.694,317.391,-94.077,174.901,29.816,155.316
C01423=1073.700,317.612,-94.106,174.903,29.819,155.316
C01424=1073.704,317.833,-94.136,174.906,29.824,155.317
C01425=1073.710,318.053,-94.165,174.908,29.828,155.318
C01426=1073.715,318.274,-94.194,174.911,29.832,155.319
C01427=1073.721,318.522,-94.227,174.914,29.836,155.319
C01428=1073.727,318.770,-94.260,174.917,29.841,155.320
C01429=1073.733,319.017,-94.293,174.920,29.846,155.321
C01430=1073.739,319.265,-94.326,174.924,29.850,155.322
C01431=1073.745,319.513,-94.359,174.926,29.855,155.323
C01432=1073.751,319.760,-94.392,174.930,29.859,155.323
C01433=1073.757,320.008,-94.425,174.932,29.864,155.324
C01434=1073.763,320.256,-94.458,174.936,29.869,155.325
C01435=1073.769,320.504,-94.491,174.938,29.873,155.326
C01436=1073.775,320.751,-94.524,174.942,29.878,155.327
C01437=1073.781,320.999,-94.557,174.945,29.883,155.327
C01438=1073.787,321.247,-94.590,174.948,29.887,155.328
C01439=1073.794,321.495,-94.623,174.951,29.892,155.329
C01440=1073.799,321.743,-94.656,174.954,29.897,155.330
C01441=1073.806,321.991,-94.689,174.957,29.901,155.331
C01442=1073.811,322.238,-94.723,174.961,29.906,155.331
C01443=1073.818,322.485,-94.756,174.963,29.911,155.332
C01444=1073.824,322.733,-94.789,174.967,29.915,155.333
C01445=1073.830,322.981,-94.822,174.970,29.920,155.334
C01446=1073.836,323.229,-94.855,174.973,29.925,155.335
C01447=1073.841,323.476,-94.888,174.976,29.929,155.336
C01448=1073.849,323.724,-94.922,174.979,29.933,155.336
C01449=1073.854,323.972,-94.955,174.982,29.939,155.337
C01450=1073.861,324.220,-94.988,174.986,29.943,155.338
C01451=1073.866,324.467,-95.021,174.988,29.948,155.339
C01452=1073.873,324.714,-95.055,174.992,29.953,155.340
C01453=1073.879,324.963,-95.089,174.995,29.957,155.341
C01454=1073.885,325.211,-95.121,174.998,29.962,155.341
C01455=1073.891,325.459,-95.155,175.001,29.966,155.342
C01456=1073.897,325.706,-95.188,175.005,29.972,155.343
C01457=1073.903,325.953,-95.221,175.007,29.976,155.344
C01458=1073.910,326.201,-95.255,175.011,29.981,155.345
C01459=1073.916,326.449,-95.289,175.014,29.985,155.346
C01460=1073.922,326.697,-95.321,175.017,29.990,155.346
C01461=1073.928,326.944,-95.355,175.020,29.995,155.347
C01462=1073.934,327.193,-95.389,175.024,29.999,155.348
C01463=1073.941,327.439,-95.423,175.027,30.004,155.349
C01464=1073.946,327.687,-95.456,175.030,30.009,155.350
C01465=1073.953,327.935,-95.490,175.034,30.014,155.351
C01466=1073.959,328.183,-95.523,175.036,30.018,155.351
C01467=1073.965,328.430,-95.557,175.040,30.023,155.352
C01468=1073.972,328.679,-95.590,175.043,30.028,155.353
C01469=1073.978,328.926,-95.624,175.046,30.033,155.354
C01470=1073.984,329.173,-95.657,175.049,30.037,155.355
C01471=1073.990,329.421,-95.691,175.053,30.042,155.356
C01472=1073.997,329.668,-95.725,175.056,30.047,155.357
C01473=1074.003,329.917,-95.759,175.059,30.052,155.357
C01474=1074.010,330.164,-95.792,175.062,30.057,155.358
C01475=1074.014,330.382,-95.822,175.065,30.060,155.359
C01476=1074.020,330.599,-95.852,175.068,30.065,155.360
C01477=1074.026,330.817,-95.881,175.071,30.069,155.361
C01478=1074.031,331.035,-95.911,175.073,30.073,155.361
C01479=1074.037,331.252,-95.941,175.076,30.077,155.362
C01480=1074.043,331.470,-95.970,175.080,30.082,155.363
C01481=1074.048,331.688,-96.001,175.082,30.086,155.364
C01482=1074.053,331.905,-96.030,175.085,30.091,155.364
C01483=1074.059,332.153,-96.064,175.088,30.095,155.365
C01484=1074.065,332.400,-96.098,175.092,30.100,155.366
C01485=1074.071,332.649,-96.132,175.094,30.105,155.367
C01486=1074.077,332.896,-96.166,175.098,30.110,155.368
C01487=1074.083,333.143,-96.200,175.101,30.115,155.369
C01488=1074.089,333.391,-96.234,175.105,30.120,155.370
C01489=1074.095,333.638,-96.268,175.107,30.125,155.371
C01490=1074.102,333.886,-96.303,175.111,30.130,155.371
C01491=1074.108,334.134,-96.337,175.114,30.135,155.372
C01492=1074.114,334.382,-96.371,175.118,30.140,155.373
C01493=1074.120,334.629,-96.405,175.120,30.144,155.374
C01494=1074.126,334.876,-96.439,175.124,30.149,155.375
C01495=1074.132,335.124,-96.474,175.127,30.154,155.376
C01496=1074.138,335.371,-96.508,175.131,30.160,155.377
C01497=1074.145,335.619,-96.542,175.133,30.164,155.378
C01498=1074.151,335.866,-96.576,175.137,30.169,155.379
C01499=1074.158,336.114,-96.610,175.140,30.174,155.380
C01500=1074.164,336.362,-96.644,175.144,30.179,155.380
C01501=1074.170,336.610,-96.679,175.147,30.184,155.381
C01502=1074.176,336.857,-96.713,175.150,30.189,155.382
C01503=1074.183,337.104,-96.748,175.153,30.194,155.383
C01504=1074.188,337.353,-96.783,175.157,30.199,155.384
C01505=1074.194,337.600,-96.817,175.160,30.204,155.385
C01506=1074.201,337.848,-96.851,175.164,30.209,155.386
C01507=1074.207,338.095,-96.885,175.166,30.215,155.387
C01508=1074.213,338.343,-96.921,175.170,30.220,155.388
C01509=1074.219,338.590,-96.955,175.173,30.225,155.389
C01510=1074.226,338.838,-96.989,175.177,30.230,155.390
C01511=1074.231,339.085,-97.024,175.180,30.235,155.390
C01512=1074.237,339.333,-97.059,175.183,30.240,155.392
C01513=1074.243,339.580,-97.093,175.186,30.245,155.392
C01514=1074.250,339.827,-97.128,175.190,30.250,155.393
C01515=1074.257,340.075,-97.162,175.193,30.256,155.394
C01516=1074.262,340.323,-97.197,175.197,30.261,155.395
C01517=1074.268,340.570,-97.232,175.200,30.266,155.396
C01518=1074.274,340.818,-97.266,175.203,30.271,155.397
C01519=1074.281,341.065,-97.301,175.206,30.276,155.398
C01520=1074.287,341.313,-97.336,175.210,30.281,155.399
C01521=1074.293,341.560,-97.371,175.213,30.286,155.400
C01522=1074.299,341.808,-97.406,175.217,30.292,155.401
C01523=1074.306,342.055,-97.441,175.220,30.297,155.402
C01524=1074.311,342.303,-97.475,175.223,30.302,155.403
C01525=1074.318,342.550,-97.510,175.227,30.307,155.404
C01526=1074.325,342.798,-97.545,175.230,30.312,155.405
C01527=1074.330,343.045,-97.580,175.234,30.318,155.406
C01528=1074.337,343.293,-97.615,175.237,30.323,155.407
C01529=1074.343,343.541,-97.650,175.241,30.328,155.408
C01530=1074.350,343.788,-97.685,175.244,30.333,155.409
C01531=1074.355,344.003,-97.715,175.247,30.337,155.409
C01532=1074.361,344.218,-97.746,175.249,30.342,155.410
C01533=1074.366,344.433,-97.776,175.253,30.347,155.411
C01534=1074.371,344.648,-97.806,175.255,30.352,155.412
C01535=1074.376,344.863,-97.838,175.259,30.356,155.413
C01536=1074.381,345.078,-97.868,175.262,30.361,155.414
C01537=1074.387,345.293,-97.899,175.264,30.365,155.415
C01538=1074.392,345.508,-97.929,175.268,30.370,155.415
C01539=1074.399,345.756,-97.964,175.271,30.375,155.416
C01540=1074.405,346.003,-98.000,175.275,30.381,155.417
C01541=1074.411,346.250,-98.034,175.277,30.386,155.418
C01542=1074.417,346.498,-98.070,175.281,30.391,155.419
C01543=1074.424,346.745,-98.105,175.284,30.396,155.420
C01544=1074.430,346.993,-98.140,175.288,30.402,155.421
C01545=1074.436,347.241,-98.175,175.291,30.407,155.422
C01546=1074.442,347.488,-98.211,175.295,30.412,155.423
C01547=1074.449,347.735,-98.246,175.298,30.418,155.424
C01548=1074.455,347.983,-98.282,175.302,30.424,155.425
C01549=1074.461,348.230,-98.317,175.305,30.429,155.426
C01550=1074.467,348.478,-98.352,175.309,30.435,155.427
C01551=1074.473,348.725,-98.388,175.312,30.440,155.428
C01552=1074.480,348.972,-98.423,175.316,30.445,155.429
C01553=1074.486,349.219,-98.459,175.319,30.451,155.430
C01554=1074.492,349.467,-98.495,175.323,30.456,155.431
C01555=1074.499,349.714,-98.530,175.326,30.462,155.433
C01556=1074.505,349.962,-98.566,175.330,30.467,155.434
C01557=1074.511,350.209,-98.602,175.333,30.472,155.435
C01558=1074.518,350.457,-98.637,175.336,30.478,155.436
C01559=1074.523,350.704,-98.672,175.340,30.483,155.437
C01560=1074.530,350.950,-98.708,175.343,30.489,155.438
C01561=1074.536,351.198,-98.744,175.347,30.494,155.439
C01562=1074.542,351.446,-98.780,175.350,30.500,155.440
C01563=1074.549,351.693,-98.815,175.354,30.505,155.441
C01564=1074.555,351.940,-98.851,175.357,30.511,155.442
C01565=1074.561,352.188,-98.887,175.361,30.516,155.443
C01566=1074.567,352.436,-98.923,175.364,30.522,155.444
C01567=1074.574,352.682,-98.958,175.368,30.527,155.445
C01568=1074.580,352.930,-98.994,175.371,30.533,155.446
C01569=1074.586,353.178,-99.030,175.375,30.539,155.447
C01570=1074.593,353.425,-99.066,175.378,30.544,155.448
C01571=1074.599,353.672,-99.102,175.382,30.550,155.449
C01572=1074.606,353.919,-99.138,175.385,30.555,155.450
C01573=1074.612,354.167,-99.174,175.389,30.561,155.451
C01574=1074.618,354.414,-99.210,175.392,30.567,155.452
C01575=1074.624,354.662,-99.246,175.396,30.572,155.453
C01576=1074.631,354.909,-99.282,175.399,30.578,155.455
C01577=1074.637,355.156,-99.318,175.403,30.584,155.456
C01578=1074.643,355.403,-99.354,175.407,30.589,155.457
C01579=1074.649,355.650,-99.391,175.411,30.595,155.458
C01580=1074.655,355.898,-99.427,175.414,30.601,155.459
C01581=1074.662,356.145,-99.463,175.418,30.607,155.460
C01582=1074.668,356.393,-99.498,175.422,30.612,155.461
C01583=1074.675,356.640,-99.535,175.425,30.618,155.462
C01584=1074.681,356.887,-99.571,175.429,30.624,155.463
C01585=1074.687,357.134,-99.607,175.432,30.629,155.464
C01586=1074.694,357.381,-99.643,175.436,30.635,155.465
C01587=1074.700,357.598,-99.676,175.438,30.640,155.466
C01588=1074.705,357.815,-99.707,175.442,30.646,155.467
C01589=1074.710,358.031,-99.739,175.445,30.651,155.468
C01590=1074.716,358.248,-99.771,175.448,30.655,155.469
C01591=1074.722,358.465,-99.803,175.452,30.661,155.470
C01592=1074.727,358.682,-99.835,175.454,30.665,155.471
C01593=1074.733,358.898,-99.867,175.458,30.671,155.472
C01594=1074.739,359.116,-99.898,175.461,30.676,155.473
C01595=1074.745,359.363,-99.935,175.465,30.682,155.474
C01596=1074.751,359.610,-99.971,175.468,30.688,155.476
C01597=1074.758,359.857,-100.008,175.472,30.693,155.477
C01598=1074.764,360.104,-100.044,175.475,30.699,155.478
C01599=1074.770,360.351,-100.081,175.479,30.705,155.479
C01600=1074.776,360.599,-100.118,175.483,30.711,155.480
C01601=1074.783,360.846,-100.154,175.486,30.717,155.481
C01602=1074.789,361.093,-100.191,175.490,30.723,155.482
C01603=1074.796,361.340,-100.227,175.493,30.729,155.483
C01604=1074.802,361.587,-100.264,175.498,30.735,155.485
C01605=1074.809,361.835,-100.301,175.501,30.741,155.486
C01606=1074.814,362.082,-100.338,175.505,30.747,155.487
C01607=1074.821,362.329,-100.375,175.508,30.753,155.488
C01608=1074.827,362.576,-100.411,175.512,30.759,155.489
C01609=1074.834,362.824,-100.448,175.515,30.765,155.490
C01610=1074.841,363.071,-100.484,175.519,30.771,155.492
C01611=1074.846,363.318,-100.521,175.523,30.777,155.493
C01612=1074.853,363.565,-100.559,175.527,30.783,155.494
C01613=1074.860,363.812,-100.595,175.531,30.789,155.495
C01614=1074.866,364.059,-100.632,175.534,30.795,155.496
C01615=1074.872,364.307,-100.669,175.538,30.801,155.497
C01616=1074.879,364.554,-100.706,175.541,30.807,155.499
C01617=1074.885,364.801,-100.743,175.546,30.813,155.500
C01618=1074.892,365.047,-100.780,175.549,30.819,155.501
C01619=1074.898,365.295,-100.817,175.553,30.825,155.502
C01620=1074.905,365.542,-100.854,175.556,30.832,155.503
C01621=1074.910,365.789,-100.892,175.560,30.838,155.505
C01622=1074.917,366.037,-100.928,175.563,30.844,155.506
C01623=1074.923,366.284,-100.966,175.568,30.850,155.507
C01624=1074.930,366.531,-101.003,175.571,30.856,155.508
C01625=1074.937,366.778,-101.040,175.575,30.863,155.509
C01626=1074.942,367.025,-101.077,175.579,30.869,155.511
C01627=1074.949,367.272,-101.114,175.582,30.875,155.512
C01628=1074.956,367.519,-101.153,175.587,30.881,155.513
C01629=1074.962,367.766,-101.189,175.590,30.888,155.514
C01630=1074.968,368.013,-101.227,175.594,30.894,155.516
C01631=1074.975,368.260,-101.264,175.597,30.900,155.517
C01632=1074.981,368.507,-101.301,175.601,30.907,155.518
C01633=1074.988,368.755,-101.339,175.605,30.913,155.519
C01634=1074.994,369.001,-101.377,175.609,30.919,155.521
C01635=1075.001,369.249,-101.413,175.612,30.925,155.522
C01636=1075.007,369.496,-101.451,175.616,30.931,155.523
C01637=1075.013,369.742,-101.488,175.621,30.938,155.524
C01638=1075.020,369.990,-101.526,175.624,30.945,155.526
C01639=1075.026,370.236,-101.564,175.628,30.951,155.527
C01640=1075.033,370.484,-101.601,175.631,30.957,155.528
C01641=1075.039,370.731,-101.639,175.636,30.964,155.529
C01642=1075.046,370.978,-101.676,175.639,30.970,155.531
C01643=1075.052,371.203,-101.710,175.643,30.976,155.532
C01644=1075.058,371.427,-101.745,175.646,30.982,155.533
C01645=1075.064,371.653,-101.779,175.650,30.987,155.534
C01646=1075.070,371.878,-101.814,175.653,30.993,155.535
C01647=1075.075,372.103,-101.848,175.656,30.999,155.536
C01648=1075.082,372.328,-101.882,175.660,31.005,155.538
C01649=1075.087,372.553,-101.917,175.663,31.011,155.539
C01650=1075.094,372.778,-101.952,175.667,31.017,155.540
C01651=1075.100,373.025,-101.989,175.671,31.023,155.541
C01652=1075.107,373.272,-102.027,175.675,31.030,155.542
C01653=1075.113,373.520,-102.065,175.679,31.036,155.544
C01654=1075.120,373.766,-102.102,175.682,31.043,155.545
C01655=1075.126,374.014,-102.140,175.687,31.050,155.546
C01656=1075.132,374.260,-102.178,175.690,31.056,155.548
C01657=1075.139,374.507,-102.217,175.694,31.063,155.549
C01658=1075.145,374.754,-102.255,175.699,31.070,155.550
C01659=1075.151,375.001,-102.293,175.702,31.076,155.552
C01660=1075.159,375.248,-102.331,175.706,31.083,155.553
C01661=1075.165,375.495,-102.369,175.710,31.090,155.554
C01662=1075.171,375.742,-102.407,175.714,31.096,155.556
C01663=1075.178,375.988,-102.445,175.717,31.103,155.557
C01664=1075.184,376.236,-102.484,175.722,31.110,155.558
C01665=1075.191,376.483,-102.522,175.725,31.117,155.560
C01666=1075.197,376.729,-102.560,175.729,31.123,155.561
C01667=1075.203,376.977,-102.598,175.734,31.130,155.563
C01668=1075.211,377.223,-102.637,175.737,31.137,155.564
C01669=1075.217,377.471,-102.675,175.741,31.143,155.565
C01670=1075.224,377.717,-102.713,175.745,31.151,155.567
C01671=1075.230,377.964,-102.751,175.749,31.157,155.568
C01672=1075.237,378.211,-102.790,175.753,31.164,155.569
C01673=1075.243,378.458,-102.828,175.757,31.171,155.571
C01674=1075.250,378.705,-102.867,175.761,31.178,155.572
C01675=1075.256,378.951,-102.905,175.765,31.184,155.574
C01676=1075.263,379.199,-102.944,175.769,31.191,155.575
C01677=1075.270,379.446,-102.982,175.773,31.199,155.576
C01678=1075.276,379.692,-103.021,175.777,31.205,155.578
C01679=1075.282,379.939,-103.059,175.781,31.212,155.579
C01680=1075.289,380.186,-103.098,175.785,31.219,155.581
C01681=1075.296,380.433,-103.137,175.789,31.226,155.582
C01682=1075.303,380.680,-103.175,175.793,31.233,155.584
C01683=1075.309,380.926,-103.213,175.797,31.240,155.585
C01684=1075.316,381.173,-103.252,175.800,31.247,155.586
C01685=1075.322,381.420,-103.291,175.805,31.254,155.588
C01686=1075.329,381.667,-103.330,175.809,31.261,155.589
C01687=1075.336,381.914,-103.369,175.813,31.268,155.591
C01688=1075.343,382.161,-103.408,175.817,31.275,155.592
C01689=1075.350,382.407,-103.446,175.821,31.282,155.593
C01690=1075.357,382.654,-103.485,175.825,31.290,155.595
C01691=1075.362,382.901,-103.524,175.830,31.297,155.596
C01692=1075.369,383.147,-103.563,175.833,31.304,155.598
C01693=1075.376,383.394,-103.602,175.838,31.311,155.599
C01694=1075.382,383.641,-103.641,175.841,31.319,155.601
C01695=1075.389,383.888,-103.680,175.846,31.326,155.602
C01696=1075.395,384.135,-103.719,175.849,31.333,155.604
C01697=1075.402,384.382,-103.758,175.854,31.340,155.605
C01698=1075.409,384.629,-103.797,175.858,31.348,155.607
C01699=1075.415,384.868,-103.835,175.861,31.354,155.608
C01700=1075.422,385.107,-103.873,175.866,31.361,155.610
C01701=1075.427,385.347,-103.911,175.870,31.369,155.611
C01702=1075.435,385.586,-103.949,175.874,31.376,155.613
C01703=1075.441,385.826,-103.987,175.878,31.383,155.614
C01704=1075.448,386.066,-104.025,175.881,31.390,155.616
C01705=1075.454,386.305,-104.064,175.886,31.397,155.617
C01706=1075.460,386.545,-104.102,175.890,31.405,155.619
C01707=1075.467,386.791,-104.141,175.894,31.412,155.620
C01708=1075.473,387.038,-104.180,175.898,31.419,155.622
C01709=1075.480,387.285,-104.220,175.902,31.427,155.623
C01710=1075.487,387.532,-104.259,175.906,31.434,155.625
C01711=1075.494,387.778,-104.299,175.911,31.442,155.626
C01712=1075.500,388.026,-104.338,175.914,31.449,155.628
C01713=1075.507,388.272,-104.378,175.919,31.456,155.629
C01714=1075.514,388.519,-104.417,175.924,31.464,155.631
C01715=1075.521,388.765,-104.457,175.927,31.471,155.633
C01716=1075.528,389.012,-104.495,175.932,31.479,155.634
C01717=1075.535,389.258,-104.535,175.935,31.487,155.636
C01718=1075.542,389.505,-104.576,175.940,31.494,155.637
C01719=1075.548,389.752,-104.614,175.945,31.502,155.639
C01720=1075.555,389.999,-104.655,175.948,31.509,155.640
C01721=1075.562,390.245,-104.694,175.953,31.517,155.642
C01722=1075.568,390.492,-104.734,175.957,31.525,155.644
C01723=1075.576,390.739,-104.773,175.961,31.532,155.645
C01724=1075.583,390.985,-104.813,175.966,31.540,155.647
C01725=1075.589,391.232,-104.853,175.969,31.548,155.648
C01726=1075.596,391.478,-104.892,175.974,31.556,155.650
C01727=1075.602,391.725,-104.932,175.979,31.563,155.652
C01728=1075.609,391.972,-104.973,175.982,31.571,155.653
C01729=1075.616,392.218,-105.012,175.987,31.579,155.655
C01730=1075.623,392.465,-105.052,175.992,31.587,155.657
C01731=1075.629,392.711,-105.092,175.995,31.594,155.658
C01732=1075.637,392.958,-105.132,176.000,31.602,155.660
C01733=1075.643,393.205,-105.173,176.004,31.610,155.662
C01734=1075.650,393.451,-105.213,176.008,31.618,155.663
C01735=1075.657,393.698,-105.253,176.013,31.626,155.665
C01736=1075.664,393.945,-105.293,176.017,31.634,155.667
C01737=1075.670,394.191,-105.333,176.021,31.642,155.668
C01738=1075.678,394.438,-105.373,176.026,31.650,155.670
C01739=1075.685,394.684,-105.414,176.030,31.658,155.672
C01740=1075.691,394.931,-105.454,176.035,31.666,155.673
C01741=1075.698,395.178,-105.494,176.039,31.674,155.675
C01742=1075.704,395.424,-105.535,176.043,31.683,155.677
C01743=1075.711,395.672,-105.575,176.048,31.691,155.679
C01744=1075.719,395.917,-105.615,176.052,31.698,155.680
C01745=1075.725,396.164,-105.655,176.056,31.707,155.682
C01746=1075.732,396.411,-105.696,176.061,31.715,155.684
C01747=1075.739,396.657,-105.737,176.066,31.723,155.685
C01748=1075.746,396.904,-105.777,176.069,31.731,155.687
C01749=1075.752,397.150,-105.817,176.074,31.739,155.689
C01750=1075.759,397.397,-105.859,176.079,31.748,155.691
C01751=1075.767,397.643,-105.898,176.083,31.756,155.692
C01752=1075.774,397.890,-105.939,176.087,31.764,155.694
C01753=1075.780,398.136,-105.980,176.092,31.773,155.696
C01754=1075.788,398.383,-106.021,176.096,31.781,155.698
C01755=1075.795,398.630,-106.061,176.101,31.789,155.699
C01756=1075.801,398.878,-106.102,176.106,31.798,155.701
C01757=1075.808,399.126,-106.143,176.109,31.806,155.703
C01758=1075.815,399.373,-106.184,176.114,31.814,155.705
C01759=1075.822,399.620,-106.226,176.119,31.823,155.707
C01760=1075.829,399.866,-106.267,176.123,31.831,155.709
C01761=1075.836,400.113,-106.307,176.128,31.840,155.710
C01762=1075.843,400.360,-106.348,176.132,31.849,155.712
C01763=1075.850,400.605,-106.389,176.137,31.857,155.714
C01764=1075.857,400.852,-106.430,176.141,31.866,155.716
C01765=1075.863,401.099,-106.471,176.146,31.874,155.718
C01766=1075.870,401.345,-106.512,176.151,31.883,155.720
C01767=1075.877,401.592,-106.554,176.155,31.892,155.721
C01768=1075.884,401.838,-106.594,176.159,31.900,155.723
C01769=1075.891,402.084,-106.636,176.164,31.909,155.725
C01770=1075.898,402.331,-106.677,176.168,31.917,155.727
C01771=1075.906,402.578,-106.718,176.173,31.926,155.729
C01772=1075.912,402.824,-106.759,176.178,31.935,155.731
C01773=1075.920,403.070,-106.800,176.183,31.944,155.733
C01774=1075.926,403.317,-106.842,176.187,31.953,155.735
C01775=1075.933,403.564,-106.883,176.192,31.961,155.736
C01776=1075.941,403.810,-106.925,176.197,31.970,155.738
C01777=1075.947,404.056,-106.965,176.201,31.979,155.740
C01778=1075.954,404.303,-107.007,176.206,31.988,155.742
C01779=1075.961,404.550,-107.048,176.210,31.997,155.744
C01780=1075.969,404.796,-107.090,176.215,32.006,155.746
C01781=1075.975,405.043,-107.132,176.219,32.015,155.748
C01782=1075.982,405.288,-107.173,176.224,32.024,155.750
C01783=1075.989,405.535,-107.214,176.229,32.032,155.752
C01784=1075.996,405.781,-107.257,176.234,32.041,155.754
C01785=1076.003,406.028,-107.298,176.238,32.051,155.756
C01786=1076.010,406.275,-107.340,176.243,32.060,155.758
C01787=1076.018,406.521,-107.382,176.248,32.069,155.760
C01788=1076.025,406.767,-107.423,176.253,32.078,155.762
C01789=1076.032,407.014,-107.466,176.257,32.087,155.764
C01790=1076.039,407.260,-107.507,176.262,32.097,155.766
C01791=1076.046,407.507,-107.549,176.267,32.105,155.768
C01792=1076.052,407.753,-107.591,176.272,32.115,155.770
C01793=1076.059,407.999,-107.633,176.276,32.124,155.772
C01794=1076.066,408.246,-107.675,176.281,32.134,155.774
C01795=1076.074,408.492,-107.717,176.287,32.143,155.776
C01796=1076.080,408.738,-107.759,176.292,32.152,155.778
C01797=1076.088,408.985,-107.800,176.297,32.162,155.780
C01798=1076.095,409.231,-107.843,176.301,32.171,155.782
C01799=1076.101,409.477,-107.885,176.306,32.180,155.784
C01800=1076.109,409.723,-107.927,176.311,32.190,155.786
C01801=1076.116,409.969,-107.970,176.316,32.199,155.788
C01802=1076.122,410.216,-108.012,176.320,32.209,155.791
C01803=1076.131,410.463,-108.054,176.325,32.219,155.793
C01804=1076.137,410.709,-108.097,176.330,32.228,155.795
C01805=1076.145,410.955,-108.139,176.336,32.237,155.797
C01806=1076.152,411.201,-108.181,176.341,32.247,155.799
C01807=1076.159,411.448,-108.224,176.345,32.257,155.801
C01808=1076.166,411.694,-108.266,176.350,32.267,155.803
C01809=1076.173,411.940,-108.308,176.355,32.276,155.805
C01810=1076.181,412.187,-108.351,176.360,32.286,155.808
C01811=1076.191,412.543,-108.412,176.368,32.300,155.811
C01812=1076.201,412.900,-108.474,176.375,32.314,155.814
C01813=1076.213,413.256,-108.536,176.382,32.328,155.817
C01814=1076.222,413.613,-108.597,176.390,32.343,155.820
